C01827=1163.106,-119.094,-41.688,178.743,5.828,149.411
C01828=1163.100,-118.844,-41.697,178.746,5.829,149.411
C01829=1163.095,-118.594,-41.706,178.747,5.829,149.410
C01830=1163.090,-118.345,-41.714,178.749,5.829,149.410
C01831=1163.084,-118.095,-41.723,178.752,5.829,149.409
C01832=1163.079,-117.845,-41.731,178.754,5.830,149.409
C01833=1163.074,-117.595,-41.740,178.755,5.830,149.408
C01834=1163.068,-117.345,-41.749,178.758,5.830,149.408
C01835=1163.063,-117.095,-41.758,178.760,5.830,149.407
C01836=1163.058,-116.846,-41.766,178.762,5.831,149.407
C01837=1163.052,-116.596,-41.775,178.763,5.831,149.406
C01838=1163.047,-116.346,-41.784,178.766,5.831,149.405
C01839=1163.042,-116.097,-41.793,178.768,5.831,149.405
C01840=1163.036,-115.846,-41.803,178.770,5.832,149.404
C01841=1163.031,-115.597,-41.812,178.772,5.831,149.404
C01842=1163.025,-115.347,-41.820,178.774,5.832,149.403
C01843=1163.020,-115.098,-41.829,178.776,5.832,149.403
C01844=1163.015,-114.848,-41.838,178.778,5.833,149.402
C01845=1163.010,-114.598,-41.847,178.780,5.832,149.402
C01846=1163.005,-114.348,-41.856,178.782,5.833,149.401
C01847=1162.999,-114.098,-41.865,178.784,5.834,149.401
C01848=1162.993,-113.849,-41.874,178.786,5.834,149.400
C01849=1162.988,-113.599,-41.883,178.789,5.834,149.399
C01850=1162.983,-113.349,-41.891,178.790,5.834,149.399
C01851=1162.977,-113.099,-41.900,178.792,5.835,149.398
C01852=1162.972,-112.849,-41.909,178.795,5.835,149.398
C01853=1162.967,-112.600,-41.918,178.797,5.835,149.397
C01854=1162.961,-112.349,-41.928,178.798,5.835,149.397
C01855=1162.956,-112.099,-41.937,178.801,5.836,149.396
C01856=1162.950,-111.850,-41.945,178.803,5.836,149.395
C01857=1162.945,-111.600,-41.954,178.805,5.836,149.395
C01858=1162.940,-111.351,-41.963,178.808,5.837,149.394
C01859=1162.935,-111.101,-41.972,178.809,5.837,149.394
C01860=1162.929,-110.851,-41.982,178.811,5.838,149.393
C01861=1162.924,-110.601,-41.991,178.813,5.838,149.393
C01862=1162.919,-110.352,-42.000,178.816,5.838,149.392
C01863=1162.914,-110.102,-42.009,178.817,5.838,149.392
C01864=1162.908,-109.852,-42.018,178.819,5.839,149.391
C01865=1162.902,-109.602,-42.027,178.821,5.838,149.390
C01866=1162.897,-109.353,-42.036,178.824,5.839,149.390
C01867=1162.892,-109.103,-42.044,178.825,5.839,149.389
C01868=1162.887,-108.853,-42.054,178.828,5.839,149.389
C01869=1162.881,-108.603,-42.064,178.830,5.840,149.388
C01870=1162.876,-108.353,-42.072,178.832,5.840,149.388
C01871=1162.870,-108.104,-42.081,178.834,5.840,149.387
C01872=1162.865,-107.854,-42.090,178.836,5.840,149.387
C01873=1162.859,-107.604,-42.100,178.838,5.841,149.386
C01874=1162.855,-107.354,-42.109,178.840,5.841,149.385
C01875=1162.849,-107.104,-42.118,178.842,5.842,149.385
C01876=1162.844,-106.855,-42.127,178.845,5.842,149.384
C01877=1162.838,-106.604,-42.137,178.847,5.842,149.384
C01878=1162.833,-106.355,-42.146,178.849,5.843,149.383
C01879=1162.828,-106.105,-42.155,178.850,5.843,149.383
C01880=1162.823,-105.856,-42.164,178.853,5.843,149.382
C01881=1162.817,-105.606,-42.173,178.855,5.843,149.382
C01882=1162.811,-105.356,-42.182,178.857,5.844,149.381
C01883=1162.807,-105.107,-42.192,178.860,5.844,149.380
C01884=1162.801,-104.857,-42.201,178.861,5.844,149.380
C01885=1162.796,-104.607,-42.210,178.863,5.845,149.379
C01886=1162.790,-104.357,-42.219,178.866,5.844,149.379
C01887=1162.785,-104.108,-42.229,178.868,5.845,149.378
C01888=1162.780,-103.858,-42.238,178.869,5.845,149.378
C01889=1162.774,-103.608,-42.247,178.872,5.846,149.377
C01890=1162.769,-103.358,-42.256,178.874,5.846,149.376
C01891=1162.764,-103.108,-42.266,178.876,5.846,149.376
C01892=1162.758,-102.859,-42.275,178.878,5.847,149.375
C01893=1162.753,-102.587,-42.285,178.880,5.847,149.375
C01894=1162.747,-102.314,-42.296,178.883,5.847,149.374
C01895=1162.741,-102.043,-42.306,178.885,5.848,149.374
C01896=1162.735,-101.770,-42.316,178.888,5.848,149.373
C01897=1162.731,-101.521,-42.325,178.889,5.848,149.372
C01898=1162.725,-101.271,-42.335,178.892,5.848,149.372
C01899=1162.720,-101.021,-42.344,178.893,5.848,149.371
C01900=1162.715,-100.772,-42.353,178.896,5.849,149.371
C01901=1162.709,-100.521,-42.363,178.898,5.850,149.370
C01902=1162.704,-100.272,-42.373,178.900,5.850,149.369
C01903=1162.698,-100.022,-42.382,178.902,5.850,149.369
C01904=1162.693,-99.772,-42.391,178.904,5.850,149.368
C01905=1162.688,-99.523,-42.401,178.906,5.851,149.368
C01906=1162.682,-99.273,-42.410,178.908,5.851,149.367
C01907=1162.677,-99.024,-42.420,178.911,5.851,149.367
C01908=1162.671,-98.773,-42.429,178.913,5.852,149.366
C01909=1162.666,-98.523,-42.438,178.915,5.851,149.365
C01910=1162.661,-98.274,-42.448,178.917,5.852,149.365
C01911=1162.655,-98.024,-42.457,178.919,5.852,149.364
C01912=1162.651,-97.775,-42.467,178.921,5.853,149.364
C01913=1162.645,-97.525,-42.476,178.924,5.853,149.363
C01914=1162.640,-97.275,-42.486,178.925,5.853,149.363
C01915=1162.634,-97.025,-42.495,178.928,5.854,149.362
C01916=1162.629,-96.775,-42.504,178.929,5.854,149.362
C01917=1162.623,-96.526,-42.514,178.932,5.854,149.361
C01918=1162.619,-96.275,-42.524,178.934,5.855,149.360
C01919=1162.613,-96.026,-42.534,178.936,5.855,149.360
C01920=1162.608,-95.776,-42.543,178.939,5.855,149.359
C01921=1162.602,-95.526,-42.553,178.941,5.856,149.359
C01922=1162.597,-95.277,-42.562,178.942,5.856,149.358
C01923=1162.591,-95.027,-42.572,178.945,5.856,149.357
C01924=1162.586,-94.777,-42.581,178.947,5.856,149.357
C01925=1162.581,-94.528,-42.591,178.949,5.857,149.357
C01926=1162.575,-94.278,-42.600,178.952,5.857,149.356
C01927=1162.570,-94.028,-42.610,178.953,5.857,149.355
C01928=1162.565,-93.778,-42.620,178.956,5.858,149.355
C01929=1162.560,-93.528,-42.630,178.957,5.858,149.354
C01930=1162.555,-93.279,-42.639,178.960,5.859,149.354
C01931=1162.549,-93.029,-42.649,178.962,5.859,149.353
C01932=1162.544,-92.780,-42.659,178.964,5.859,149.352
C01933=1162.538,-92.529,-42.668,178.967,5.859,149.352
C01934=1162.533,-92.280,-42.678,178.969,5.860,149.351
C01935=1162.527,-92.030,-42.687,178.970,5.860,149.351
C01936=1162.523,-91.780,-42.697,178.973,5.860,149.350
C01937=1162.518,-91.530,-42.707,178.975,5.860,149.350
C01938=1162.512,-91.280,-42.717,178.977,5.861,149.349
C01939=1162.507,-91.031,-42.726,178.979,5.862,149.348
C01940=1162.501,-90.782,-42.737,178.981,5.862,149.348
C01941=1162.496,-90.532,-42.746,178.984,5.862,149.347
C01942=1162.491,-90.281,-42.756,178.986,5.863,149.347
C01943=1162.485,-90.031,-42.766,178.988,5.862,149.346
C01944=1162.480,-89.782,-42.775,178.990,5.863,149.346
C01945=1162.475,-89.533,-42.785,178.992,5.863,149.345
C01946=1162.469,-89.283,-42.794,178.994,5.863,149.344
C01947=1162.464,-89.033,-42.805,178.997,5.864,149.344
C01948=1162.459,-88.783,-42.815,178.999,5.864,149.343
C01949=1162.454,-88.533,-42.824,179.001,5.865,149.343
C01950=1162.448,-88.283,-42.834,179.003,5.865,149.342
C01951=1162.443,-88.034,-42.844,179.005,5.865,149.341
C01952=1162.438,-87.785,-42.854,179.007,5.866,149.341
C01953=1162.432,-87.534,-42.864,179.010,5.866,149.340
C01954=1162.427,-87.285,-42.874,179.012,5.866,149.340
C01955=1162.422,-87.035,-42.884,179.014,5.867,149.339
C01956=1162.416,-86.785,-42.893,179.017,5.867,149.339
C01957=1162.411,-86.536,-42.903,179.018,5.867,149.338
C01958=1162.406,-86.285,-42.913,179.021,5.868,149.337
C01959=1162.401,-86.036,-42.924,179.022,5.868,149.337
C01960=1162.395,-85.786,-42.933,179.025,5.868,149.336
C01961=1162.390,-85.536,-42.943,179.027,5.869,149.336
C01962=1162.385,-85.286,-42.953,179.029,5.869,149.335
C01963=1162.380,-85.037,-42.963,179.032,5.869,149.335
C01964=1162.374,-84.787,-42.973,179.034,5.870,149.334
C01965=1162.368,-84.537,-42.983,179.036,5.869,149.333
C01966=1162.364,-84.288,-42.992,179.038,5.870,149.333
C01967=1162.359,-84.038,-43.003,179.040,5.871,149.332
C01968=1162.353,-83.788,-43.013,179.042,5.871,149.332
C01969=1162.348,-83.539,-43.023,179.044,5.871,149.331
C01970=1162.343,-83.288,-43.032,179.047,5.872,149.330
C01971=1162.337,-83.039,-43.043,179.049,5.872,149.330
C01972=1162.332,-82.789,-43.053,179.051,5.873,149.330
C01973=1162.327,-82.540,-43.063,179.054,5.873,149.329
C01974=1162.322,-82.290,-43.073,179.055,5.873,149.328
C01975=1162.316,-82.040,-43.083,179.058,5.873,149.328
C01976=1162.311,-81.791,-43.094,179.060,5.874,149.327
C01977=1162.305,-81.541,-43.102,179.062,5.874,149.326
C01978=1162.300,-81.290,-43.113,179.064,5.874,149.326
C01979=1162.295,-81.041,-43.123,179.066,5.875,149.325
C01980=1162.289,-80.791,-43.133,179.069,5.875,149.325
C01981=1162.285,-80.541,-43.143,179.071,5.876,149.324
C01982=1162.279,-80.292,-43.154,179.073,5.876,149.324
C01983=1162.274,-80.042,-43.164,179.075,5.876,149.323
C01984=1162.268,-79.793,-43.174,179.078,5.876,149.322
C01985=1162.263,-79.543,-43.185,179.080,5.877,149.322
C01986=1162.258,-79.293,-43.194,179.081,5.877,149.321
C01987=1162.253,-79.044,-43.204,179.084,5.877,149.321
C01988=1162.248,-78.794,-43.215,179.086,5.878,149.320
C01989=1162.242,-78.544,-43.225,179.088,5.878,149.319
C01990=1162.236,-78.294,-43.235,179.091,5.879,149.319
C01991=1162.231,-78.044,-43.245,179.093,5.879,149.318
C01992=1162.226,-77.794,-43.255,179.095,5.880,149.318
C01993=1162.221,-77.545,-43.265,179.098,5.879,149.317
C01994=1162.216,-77.295,-43.276,179.100,5.880,149.317
C01995=1162.210,-77.045,-43.286,179.102,5.881,149.316
C01996=1162.205,-76.795,-43.296,179.104,5.881,149.315
C01997=1162.199,-76.524,-43.307,179.107,5.881,149.315
C01998=1162.194,-76.253,-43.319,179.109,5.882,149.314
C01999=1162.188,-75.983,-43.330,179.112,5.882,149.314
C02000=1162.182,-75.711,-43.341,179.114,5.883,149.313
C02001=1162.176,-75.461,-43.352,179.116,5.883,149.312
C02002=1162.171,-75.211,-43.362,179.118,5.883,149.312
C02003=1162.166,-74.962,-43.372,179.121,5.884,149.311
C02004=1162.160,-74.712,-43.383,179.122,5.884,149.311
C02005=1162.155,-74.462,-43.393,179.125,5.884,149.310
C02006=1162.150,-74.213,-43.403,179.127,5.885,149.309
C02007=1162.145,-73.962,-43.413,179.130,5.885,149.309
C02008=1162.140,-73.713,-43.424,179.131,5.885,149.308
C02009=1162.134,-73.463,-43.434,179.134,5.886,149.308
C02010=1162.129,-73.213,-43.444,179.136,5.886,149.307
C02011=1162.124,-72.964,-43.455,179.138,5.886,149.307
C02012=1162.118,-72.715,-43.465,179.140,5.887,149.306
C02013=1162.113,-72.464,-43.476,179.143,5.888,149.305
C02014=1162.108,-72.215,-43.486,179.145,5.888,149.305
C02015=1162.103,-71.965,-43.497,179.147,5.888,149.304
C02016=1162.097,-71.715,-43.507,179.150,5.888,149.304
C02017=1162.092,-71.465,-43.518,179.152,5.889,149.303
C02018=1162.087,-71.216,-43.529,179.154,5.889,149.302
C02019=1162.081,-70.966,-43.539,179.156,5.890,149.302
C02020=1162.076,-70.716,-43.549,179.159,5.890,149.301
C02021=1162.071,-70.467,-43.560,179.161,5.891,149.301
C02022=1162.066,-70.216,-43.570,179.163,5.890,149.300
C02023=1162.060,-69.967,-43.580,179.165,5.891,149.299
C02024=1162.055,-69.717,-43.592,179.167,5.892,149.299
C02025=1162.050,-69.468,-43.602,179.169,5.891,149.298
C02026=1162.044,-69.218,-43.612,179.172,5.892,149.298
C02027=1162.039,-68.968,-43.623,179.174,5.893,149.297
C02028=1162.034,-68.719,-43.634,179.177,5.893,149.297
C02029=1162.029,-68.469,-43.644,179.179,5.893,149.296
C02030=1162.023,-68.219,-43.654,179.181,5.894,149.295
C02031=1162.018,-67.969,-43.665,179.183,5.894,149.295
C02032=1162.013,-67.720,-43.676,179.186,5.895,149.294
C02033=1162.008,-67.470,-43.686,179.188,5.895,149.294
C02034=1162.002,-67.220,-43.697,179.190,5.895,149.293
C02035=1161.997,-66.970,-43.707,179.193,5.896,149.292
C02036=1161.992,-66.721,-43.718,179.194,5.896,149.292
C02037=1161.987,-66.471,-43.729,179.197,5.896,149.291
C02038=1161.981,-66.221,-43.739,179.199,5.897,149.291
C02039=1161.977,-65.972,-43.750,179.202,5.897,149.290
C02040=1161.971,-65.722,-43.760,179.203,5.897,149.290
C02041=1161.965,-65.471,-43.772,179.206,5.898,149.289
C02042=1161.960,-65.222,-43.782,179.208,5.899,149.288
C02043=1161.955,-64.972,-43.793,179.210,5.899,149.288
C02044=1161.950,-64.723,-43.803,179.212,5.899,149.287
C02045=1161.945,-64.473,-43.815,179.215,5.900,149.287
C02046=1161.939,-64.224,-43.825,179.217,5.900,149.286
C02047=1161.935,-63.974,-43.836,179.219,5.901,149.285
C02048=1161.929,-63.724,-43.846,179.222,5.900,149.285
C02049=1161.924,-63.474,-43.857,179.224,5.901,149.284
C02050=1161.918,-63.225,-43.868,179.226,5.902,149.284
C02051=1161.913,-62.975,-43.879,179.229,5.902,149.283
C02052=1161.908,-62.726,-43.890,179.231,5.902,149.282
C02053=1161.903,-62.475,-43.900,179.233,5.903,149.282
C02054=1161.897,-62.226,-43.911,179.236,5.903,149.281
C02055=1161.892,-61.976,-43.922,179.238,5.904,149.281
C02056=1161.887,-61.727,-43.932,179.240,5.904,149.280
C02057=1161.881,-61.477,-43.944,179.242,5.904,149.280
C02058=1161.876,-61.227,-43.955,179.245,5.905,149.279
C02059=1161.871,-60.978,-43.965,179.247,5.906,149.278
C02060=1161.866,-60.727,-43.976,179.249,5.906,149.278
C02061=1161.861,-60.478,-43.987,179.251,5.906,149.277
C02062=1161.855,-60.228,-43.998,179.254,5.906,149.276
C02063=1161.850,-59.978,-44.009,179.256,5.907,149.276
C02064=1161.845,-59.729,-44.020,179.259,5.908,149.275
C02065=1161.840,-59.479,-44.031,179.260,5.908,149.275
C02066=1161.834,-59.230,-44.041,179.263,5.908,149.274
C02067=1161.829,-58.980,-44.053,179.265,5.909,149.274
C02068=1161.823,-58.730,-44.063,179.268,5.909,149.273
C02069=1161.819,-58.480,-44.075,179.269,5.909,149.272
C02070=1161.814,-58.230,-44.085,179.272,5.910,149.272
C02071=1161.808,-57.981,-44.096,179.274,5.910,149.271
C02072=1161.803,-57.731,-44.107,179.277,5.911,149.271
C02073=1161.798,-57.481,-44.118,179.279,5.912,149.270
C02074=1161.792,-57.232,-44.129,179.281,5.911,149.269
C02075=1161.788,-56.982,-44.140,179.283,5.912,149.269
C02076=1161.782,-56.733,-44.152,179.286,5.912,149.268
C02077=1161.777,-56.482,-44.162,179.288,5.913,149.268
C02078=1161.772,-56.233,-44.173,179.291,5.914,149.267
C02079=1161.766,-55.983,-44.184,179.292,5.914,149.267
C02080=1161.761,-55.733,-44.195,179.295,5.914,149.266
C02081=1161.756,-55.484,-44.207,179.297,5.915,149.265
C02082=1161.751,-55.234,-44.217,179.300,5.915,149.265
C02083=1161.745,-54.984,-44.229,179.301,5.915,149.264
C02084=1161.741,-54.735,-44.240,179.304,5.916,149.263
C02085=1161.735,-54.485,-44.250,179.306,5.916,149.263
C02086=1161.730,-54.235,-44.262,179.309,5.917,149.262
C02087=1161.725,-53.986,-44.274,179.311,5.918,149.262
C02088=1161.719,-53.736,-44.284,179.313,5.917,149.261
C02089=1161.714,-53.486,-44.296,179.315,5.918,149.261
C02090=1161.709,-53.236,-44.307,179.318,5.918,149.260
C02091=1161.703,-52.987,-44.317,179.320,5.919,149.259
C02092=1161.698,-52.737,-44.329,179.323,5.920,149.259
C02093=1161.693,-52.487,-44.340,179.325,5.920,149.258
C02094=1161.688,-52.238,-44.351,179.327,5.920,149.258
C02095=1161.682,-51.988,-44.362,179.329,5.921,149.257
C02096=1161.678,-51.738,-44.374,179.332,5.921,149.256
C02097=1161.672,-51.489,-44.385,179.334,5.922,149.256
C02098=1161.667,-51.239,-44.396,179.337,5.922,149.255
C02099=1161.662,-50.989,-44.407,179.339,5.922,149.255
C02100=1161.657,-50.739,-44.419,179.341,5.923,149.254
C02101=1161.650,-50.469,-44.431,179.343,5.924,149.254
C02102=1161.646,-50.199,-44.443,179.346,5.924,149.253
C02103=1161.640,-49.928,-44.455,179.349,5.924,149.252
C02104=1161.634,-49.658,-44.467,179.351,5.925,149.251
C02105=1161.628,-49.408,-44.479,179.354,5.926,149.251
C02106=1161.624,-49.158,-44.491,179.356,5.926,149.250
C02107=1161.618,-48.909,-44.501,179.358,5.927,149.250
C02108=1161.613,-48.659,-44.513,179.361,5.926,149.249
C02109=1161.608,-48.409,-44.524,179.363,5.927,149.249
C02110=1161.603,-48.159,-44.536,179.365,5.928,149.248
C02111=1161.597,-47.910,-44.547,179.368,5.928,149.247
C02112=1161.592,-47.660,-44.559,179.370,5.929,149.247
C02113=1161.587,-47.411,-44.570,179.372,5.929,149.246
C02114=1161.581,-47.160,-44.581,179.374,5.929,149.246
C02115=1161.576,-46.911,-44.592,179.377,5.930,149.245
C02116=1161.571,-46.661,-44.604,179.379,5.931,149.244
C02117=1161.566,-46.411,-44.615,179.382,5.931,149.244
C02118=1161.561,-46.162,-44.627,179.384,5.932,149.243
C02119=1161.555,-45.913,-44.638,179.386,5.932,149.243
C02120=1161.550,-45.663,-44.650,179.388,5.932,149.242
C02121=1161.545,-45.413,-44.661,179.391,5.933,149.242
C02122=1161.540,-45.163,-44.673,179.393,5.933,149.241
C02123=1161.535,-44.913,-44.684,179.395,5.934,149.240
C02124=1161.529,-44.664,-44.696,179.398,5.935,149.240
C02125=1161.524,-44.415,-44.707,179.400,5.935,149.239
C02126=1161.519,-44.165,-44.719,179.402,5.935,149.238
C02127=1161.514,-43.915,-44.730,179.405,5.935,149.238
C02128=1161.509,-43.665,-44.742,179.407,5.936,149.237
C02129=1161.502,-43.415,-44.753,179.410,5.937,149.237
C02130=1161.498,-43.166,-44.764,179.412,5.937,149.236
C02131=1161.492,-42.916,-44.776,179.415,5.938,149.235
C02132=1161.488,-42.667,-44.788,179.417,5.939,149.235
C02133=1161.483,-42.417,-44.800,179.419,5.938,149.234
C02134=1161.478,-42.167,-44.811,179.421,5.939,149.234
C02135=1161.472,-41.918,-44.823,179.424,5.939,149.233
C02136=1161.466,-41.668,-44.835,179.426,5.940,149.233
C02137=1161.462,-41.418,-44.846,179.429,5.941,149.232
C02138=1161.456,-41.168,-44.858,179.431,5.941,149.231
C02139=1161.452,-40.919,-44.869,179.434,5.942,149.231
C02140=1161.446,-40.669,-44.881,179.435,5.942,149.230
C02141=1161.441,-40.419,-44.893,179.438,5.942,149.230
C02142=1161.435,-40.170,-44.904,179.440,5.943,149.229
C02143=1161.430,-39.920,-44.916,179.443,5.944,149.228
C02144=1161.425,-39.670,-44.928,179.445,5.944,149.228
C02145=1161.420,-39.420,-44.939,179.448,5.945,149.227
C02146=1161.414,-39.171,-44.951,179.450,5.945,149.226
C02147=1161.409,-38.921,-44.963,179.452,5.946,149.226
C02148=1161.405,-38.672,-44.975,179.454,5.946,149.225
C02149=1161.399,-38.422,-44.987,179.457,5.946,149.225
C02150=1161.393,-38.172,-44.998,179.459,5.947,149.224
C02151=1161.388,-37.923,-45.009,179.461,5.948,149.224
C02152=1161.383,-37.673,-45.021,179.464,5.948,149.223
C02153=1161.378,-37.423,-45.033,179.466,5.949,149.222
C02154=1161.373,-37.174,-45.045,179.469,5.949,149.222
C02155=1161.368,-36.924,-45.057,179.471,5.950,149.221
C02156=1161.362,-36.674,-45.069,179.473,5.950,149.221
C02157=1161.358,-36.424,-45.080,179.475,5.950,149.220
C02158=1161.352,-36.174,-45.092,179.478,5.951,149.219
C02159=1161.347,-35.925,-45.105,179.480,5.952,149.219
C02160=1161.342,-35.675,-45.117,179.483,5.952,149.218
C02161=1161.336,-35.426,-45.128,179.486,5.953,149.218
C02162=1161.331,-35.176,-45.139,179.488,5.953,149.217
C02163=1161.326,-34.927,-45.152,179.490,5.954,149.216
C02164=1161.320,-34.677,-45.164,179.493,5.955,149.216
C02165=1161.316,-34.428,-45.175,179.495,5.954,149.215
C02166=1161.310,-34.178,-45.187,179.497,5.955,149.215
C02167=1161.305,-33.928,-45.200,179.500,5.955,149.214
C02168=1161.300,-33.678,-45.212,179.502,5.956,149.214
C02169=1161.295,-33.429,-45.223,179.504,5.957,149.213
C02170=1161.290,-33.179,-45.235,179.507,5.957,149.212
C02171=1161.285,-32.929,-45.247,179.509,5.958,149.212
C02172=1161.279,-32.679,-45.259,179.511,5.959,149.211
C02173=1161.274,-32.430,-45.272,179.514,5.959,149.211
C02174=1161.269,-32.181,-45.283,179.516,5.960,149.210
C02175=1161.264,-31.931,-45.295,179.519,5.960,149.209
C02176=1161.259,-31.681,-45.308,179.521,5.960,149.209
C02177=1161.253,-31.431,-45.320,179.523,5.961,149.208
C02178=1161.248,-31.181,-45.331,179.526,5.961,149.208
C02179=1161.243,-30.932,-45.344,179.528,5.962,149.207
C02180=1161.238,-30.682,-45.355,179.531,5.962,149.206
C02181=1161.233,-30.433,-45.367,179.533,5.963,149.206
C02182=1161.227,-30.183,-45.380,179.535,5.964,149.205
C02183=1161.222,-29.933,-45.392,179.538,5.964,149.205
C02184=1161.217,-29.684,-45.404,179.540,5.965,149.204
C02185=1161.211,-29.434,-45.416,179.543,5.966,149.204
C02186=1161.207,-29.185,-45.428,179.545,5.966,149.203
C02187=1161.202,-28.935,-45.440,179.548,5.967,149.202
C02188=1161.196,-28.685,-45.452,179.550,5.967,149.202
C02189=1161.191,-28.436,-45.465,179.552,5.967,149.201
C02190=1161.186,-28.186,-45.476,179.554,5.968,149.200
C02191=1161.181,-27.937,-45.489,179.557,5.968,149.200
C02192=1161.175,-27.687,-45.501,179.559,5.969,149.199
C02193=1161.170,-27.437,-45.514,179.562,5.969,149.199
C02194=1161.165,-27.187,-45.525,179.564,5.970,149.198
C02195=1161.160,-26.937,-45.538,179.567,5.971,149.197
C02196=1161.155,-26.688,-45.550,179.569,5.971,149.197
C02197=1161.150,-26.438,-45.562,179.571,5.972,149.196
C02198=1161.145,-26.188,-45.574,179.574,5.973,149.196
C02199=1161.140,-25.939,-45.587,179.576,5.973,149.195
C02200=1161.134,-25.689,-45.599,179.579,5.974,149.194
C02201=1161.129,-25.440,-45.611,179.581,5.974,149.194
C02202=1161.124,-25.190,-45.623,179.584,5.975,149.193
C02203=1161.119,-24.941,-45.636,179.586,5.976,149.193
C02204=1161.113,-24.691,-45.648,179.589,5.976,149.192
C02205=1161.108,-24.421,-45.661,179.591,5.977,149.192
C02206=1161.102,-24.151,-45.676,179.593,5.977,149.191
C02207=1161.097,-23.881,-45.688,179.596,5.978,149.190
C02208=1161.091,-23.611,-45.701,179.599,5.978,149.190
C02209=1161.086,-23.362,-45.714,179.601,5.979,149.189
C02210=1161.081,-23.112,-45.726,179.604,5.979,149.188
C02211=1161.076,-22.862,-45.738,179.606,5.980,149.188
C02212=1161.070,-22.613,-45.751,179.609,5.981,149.187
C02213=1161.065,-22.364,-45.763,179.611,5.981,149.187
C02214=1161.060,-22.113,-45.776,179.613,5.982,149.186
C02215=1161.055,-21.864,-45.788,179.616,5.982,149.185
C02216=1161.050,-21.614,-45.801,179.618,5.983,149.185
C02217=1161.045,-21.365,-45.813,179.621,5.984,149.184
C02218=1161.039,-21.115,-45.826,179.623,5.984,149.184
C02219=1161.034,-20.866,-45.839,179.626,5.985,149.183
C02220=1161.028,-20.616,-45.850,179.628,5.986,149.183
C02221=1161.024,-20.366,-45.863,179.631,5.986,149.182
C02222=1161.019,-20.116,-45.876,179.633,5.987,149.181
C02223=1161.014,-19.867,-45.889,179.635,5.987,149.181
C02224=1161.008,-19.617,-45.900,179.638,5.988,149.180
C02225=1161.003,-19.368,-45.913,179.640,5.988,149.180
C02226=1160.999,-19.118,-45.926,179.642,5.988,149.179
C02227=1160.993,-18.868,-45.938,179.644,5.989,149.178
C02228=1160.988,-18.618,-45.951,179.647,5.989,149.178
C02229=1160.982,-18.369,-45.964,179.649,5.990,149.177
C02230=1160.977,-18.120,-45.976,179.652,5.991,149.176
C02231=1160.972,-17.870,-45.989,179.654,5.991,149.176
C02232=1160.967,-17.620,-46.001,179.657,5.992,149.175
C02233=1160.962,-17.370,-46.014,179.659,5.993,149.175
C02234=1160.957,-17.121,-46.026,179.662,5.993,149.174
C02235=1160.952,-16.872,-46.039,179.664,5.994,149.174
C02236=1160.946,-16.621,-46.053,179.666,5.994,149.173
C02237=1160.941,-16.372,-46.065,179.669,5.995,149.172
C02238=1160.936,-16.122,-46.077,179.671,5.996,149.172
C02239=1160.931,-15.873,-46.090,179.674,5.996,149.171
C02240=1160.926,-15.623,-46.102,179.676,5.997,149.171
C02241=1160.921,-15.373,-46.115,179.679,5.997,149.170
C02242=1160.915,-15.124,-46.128,179.681,5.998,149.170
C02243=1160.910,-14.874,-46.141,179.684,5.999,149.169
C02244=1160.905,-14.625,-46.154,179.686,5.999,149.168
C02245=1160.900,-14.375,-46.167,179.688,6.000,149.168
C02246=1160.895,-14.125,-46.178,179.691,6.000,149.167
C02247=1160.889,-13.876,-46.192,179.693,6.001,149.166
C02248=1160.884,-13.626,-46.204,179.696,6.002,149.166
C02249=1160.879,-13.376,-46.217,179.698,6.002,149.165
C02250=1160.874,-13.127,-46.230,179.701,6.003,149.165
C02251=1160.869,-12.877,-46.243,179.703,6.004,149.164
C02252=1160.864,-12.627,-46.256,179.706,6.004,149.163
C02253=1160.859,-12.378,-46.269,179.708,6.005,149.163
C02254=1160.854,-12.129,-46.281,179.711,6.006,149.162
C02255=1160.848,-11.879,-46.294,179.713,6.007,149.162
C02256=1160.843,-11.629,-46.307,179.716,6.007,149.161
C02257=1160.838,-11.380,-46.320,179.719,6.008,149.160
C02258=1160.833,-11.130,-46.333,179.721,6.009,149.160
C02259=1160.828,-10.880,-46.346,179.723,6.009,149.159
C02260=1160.823,-10.631,-46.359,179.726,6.010,149.159
C02261=1160.818,-10.381,-46.371,179.728,6.010,149.158
C02262=1160.812,-10.131,-46.385,179.730,6.011,149.158
C02263=1160.807,-9.882,-46.397,179.733,6.012,149.157
C02264=1160.802,-9.632,-46.410,179.735,6.012,149.157
C02265=1160.797,-9.382,-46.424,179.738,6.013,149.156
C02266=1160.792,-9.133,-46.436,179.741,6.013,149.155
C02267=1160.787,-8.884,-46.450,179.743,6.014,149.155
C02268=1160.782,-8.634,-46.463,179.745,6.015,149.154
C02269=1160.777,-8.384,-46.476,179.748,6.015,149.154
C02270=1160.771,-8.135,-46.488,179.750,6.016,149.153
C02271=1160.766,-7.885,-46.502,179.752,6.017,149.152
C02272=1160.761,-7.635,-46.514,179.755,6.017,149.152
C02273=1160.756,-7.385,-46.527,179.757,6.018,149.151
C02274=1160.751,-7.136,-46.541,179.760,6.018,149.151
C02275=1160.746,-6.887,-46.554,179.762,6.019,149.150
C02276=1160.741,-6.637,-46.567,179.765,6.020,149.149
C02277=1160.735,-6.387,-46.580,179.767,6.020,149.149
C02278=1160.730,-6.138,-46.593,179.770,6.021,149.148
C02279=1160.725,-5.888,-46.606,179.772,6.021,149.148
C02280=1160.720,-5.638,-46.619,179.775,6.023,149.147
C02281=1160.715,-5.389,-46.633,179.778,6.023,149.146
C02282=1160.710,-5.139,-46.646,179.780,6.024,149.146
C02283=1160.705,-4.890,-46.658,179.782,6.025,149.145
C02284=1160.699,-4.640,-46.672,179.785,6.025,149.145
C02285=1160.694,-4.390,-46.685,179.787,6.026,149.144
C02286=1160.689,-4.141,-46.699,179.789,6.027,149.144
C02287=1160.684,-3.891,-46.711,179.792,6.027,149.143
C02288=1160.678,-3.642,-46.725,179.795,6.028,149.142
C02289=1160.674,-3.392,-46.738,179.797,6.028,149.142
C02290=1160.668,-3.143,-46.751,179.800,6.029,149.141
C02291=1160.664,-2.893,-46.764,179.802,6.030,149.141
C02292=1160.658,-2.643,-46.778,179.804,6.030,149.140
C02293=1160.654,-2.394,-46.791,179.807,6.031,149.139
C02294=1160.649,-2.144,-46.804,179.810,6.032,149.139
C02295=1160.643,-1.894,-46.817,179.812,6.033,149.138
C02296=1160.638,-1.645,-46.831,179.815,6.033,149.138
C02297=1160.633,-1.396,-46.844,179.817,6.034,149.137
C02298=1160.627,-1.145,-46.858,179.820,6.035,149.136
C02299=1160.623,-0.897,-46.871,179.822,6.035,149.136
C02300=1160.617,-0.646,-46.884,179.824,6.036,149.135
C02301=1160.612,-0.397,-46.897,179.827,6.036,149.135
C02302=1160.607,-0.147,-46.911,179.829,6.037,149.134
C02303=1160.602,0.102,-46.924,179.832,6.038,149.133
C02304=1160.597,0.352,-46.937,179.834,6.039,149.133
C02305=1160.592,0.601,-46.951,179.837,6.039,149.132
C02306=1160.587,0.851,-46.964,179.839,6.041,149.132
C02307=1160.581,1.100,-46.978,179.842,6.041,149.131
C02308=1160.577,1.350,-46.991,179.844,6.042,149.131
C02309=1160.571,1.619,-47.006,179.847,6.042,149.130
C02310=1160.565,1.889,-47.020,179.850,6.043,149.129
C02311=1160.560,2.158,-47.035,179.853,6.044,149.129
C02312=1160.555,2.428,-47.050,179.855,6.045,149.128
C02313=1160.549,2.677,-47.063,179.858,6.045,149.127
C02314=1160.545,2.927,-47.076,179.860,6.046,149.127
C02315=1160.539,3.176,-47.090,179.862,6.047,149.126
C02316=1160.534,3.426,-47.104,179.865,6.047,149.126
C02317=1160.529,3.675,-47.116,179.867,6.048,149.125
C02318=1160.524,3.925,-47.131,179.870,6.048,149.124
C02319=1160.518,4.175,-47.144,179.873,6.050,149.124
C02320=1160.514,4.424,-47.158,179.875,6.050,149.123
C02321=1160.508,4.674,-47.171,179.878,6.051,149.123
C02322=1160.503,4.923,-47.185,179.880,6.052,149.122
C02323=1160.499,5.173,-47.199,179.882,6.053,149.122
C02324=1160.493,5.422,-47.212,179.885,6.053,149.121
C02325=1160.488,5.672,-47.226,179.888,6.053,149.120
C02326=1160.483,5.921,-47.239,179.890,6.054,149.120
C02327=1160.478,6.171,-47.253,179.893,6.055,149.119
C02328=1160.473,6.421,-47.267,179.895,6.056,149.119
C02329=1160.468,6.670,-47.280,179.898,6.057,149.118
C02330=1160.463,6.920,-47.294,179.900,6.058,149.118
C02331=1160.457,7.169,-47.307,179.903,6.058,149.117
C02332=1160.453,7.419,-47.321,179.905,6.059,149.116
C02333=1160.448,7.669,-47.335,179.908,6.059,149.116
C02334=1160.442,7.918,-47.349,179.910,6.060,149.115
C02335=1160.437,8.168,-47.363,179.913,6.061,149.115
C02336=1160.432,8.417,-47.376,179.915,6.062,149.114
C02337=1160.427,8.667,-47.390,179.918,6.063,149.113
C02338=1160.422,8.917,-47.404,179.920,6.063,149.113
C02339=1160.416,9.166,-47.418,179.923,6.064,149.112
C02340=1160.412,9.416,-47.431,179.925,6.064,149.112
C02341=1160.407,9.665,-47.445,179.927,6.065,149.111
C02342=1160.401,9.914,-47.459,179.931,6.067,149.110
C02343=1160.396,10.165,-47.473,179.933,6.067,149.110
C02344=1160.390,10.414,-47.487,179.935,6.068,149.109
C02345=1160.386,10.663,-47.500,179.938,6.069,149.109
C02346=1160.381,10.913,-47.515,179.940,6.069,149.108
C02347=1160.375,11.162,-47.528,179.942,6.070,149.108
C02348=1160.370,11.412,-47.542,179.946,6.071,149.107
C02349=1160.366,11.662,-47.556,179.948,6.072,149.107
C02350=1160.360,11.911,-47.570,179.951,6.072,149.106
C02351=1160.356,12.160,-47.584,179.953,6.073,149.105
C02352=1160.350,12.411,-47.597,179.955,6.074,149.105
C02353=1160.345,12.660,-47.611,179.958,6.074,149.104
C02354=1160.340,12.909,-47.626,179.961,6.076,149.104
C02355=1160.335,13.159,-47.640,179.963,6.076,149.103
C02356=1160.330,13.409,-47.654,179.966,6.077,149.102
C02357=1160.325,13.658,-47.668,179.968,6.078,149.102
C02358=1160.320,13.908,-47.681,179.970,6.078,149.101
C02359=1160.315,14.158,-47.695,179.973,6.079,149.101
C02360=1160.309,14.407,-47.709,179.976,6.081,149.100
C02361=1160.305,14.656,-47.724,179.978,6.081,149.100
C02362=1160.300,14.906,-47.738,179.981,6.082,149.099
C02363=1160.295,15.156,-47.752,179.983,6.082,149.098
C02364=1160.289,15.405,-47.766,179.986,6.083,149.098
C02365=1160.284,15.654,-47.780,179.988,6.084,149.097
C02366=1160.279,15.904,-47.795,179.991,6.085,149.097
C02367=1160.274,16.153,-47.808,179.994,6.086,149.096
C02368=1160.268,16.403,-47.822,179.996,6.086,149.095
C02369=1160.263,16.653,-47.836,179.998,6.087,149.095
C02370=1160.258,16.903,-47.851,-179.999,6.087,149.094
C02371=1160.254,17.152,-47.864,-179.996,6.089,149.094
C02372=1160.249,17.401,-47.878,-179.994,6.090,149.093
C02373=1160.244,17.651,-47.892,-179.991,6.090,149.093
C02374=1160.239,17.901,-47.907,-179.989,6.091,149.092
C02375=1160.234,18.150,-47.921,-179.987,6.092,149.092
C02376=1160.228,18.399,-47.935,-179.983,6.093,149.091
C02377=1160.223,18.649,-47.949,-179.981,6.094,149.090
C02378=1160.218,18.899,-47.963,-179.979,6.094,149.090
C02379=1160.213,19.149,-47.978,-179.976,6.095,149.089
C02380=1160.208,19.398,-47.992,-179.974,6.096,149.089
C02381=1160.203,19.647,-48.007,-179.970,6.097,149.088
C02382=1160.198,19.896,-48.021,-179.968,6.098,149.087
C02383=1160.193,20.146,-48.036,-179.966,6.098,149.087
C02384=1160.188,20.396,-48.050,-179.964,6.099,149.086
C02385=1160.183,20.646,-48.064,-179.961,6.099,149.086
C02386=1160.177,20.895,-48.078,-179.958,6.101,149.085
C02387=1160.172,21.145,-48.093,-179.955,6.102,149.084
C02388=1160.167,21.394,-48.107,-179.953,6.102,149.084
C02389=1160.162,21.644,-48.121,-179.951,6.103,149.083
C02390=1160.157,21.894,-48.135,-179.948,6.104,149.083
C02391=1160.153,22.143,-48.150,-179.945,6.105,149.082
C02392=1160.147,22.392,-48.164,-179.943,6.106,149.082
C02393=1160.142,22.641,-48.179,-179.940,6.106,149.081
C02394=1160.137,22.891,-48.193,-179.938,6.107,149.081
C02395=1160.132,23.141,-48.207,-179.935,6.108,149.080
C02396=1160.126,23.391,-48.222,-179.933,6.109,149.079
C02397=1160.122,23.640,-48.237,-179.930,6.110,149.079
C02398=1160.117,23.890,-48.251,-179.928,6.110,149.078
C02399=1160.111,24.139,-48.265,-179.925,6.112,149.078
C02400=1160.106,24.388,-48.279,-179.923,6.113,149.077
C02401=1160.102,24.638,-48.294,-179.920,6.113,149.077
C02402=1160.097,24.887,-48.309,-179.918,6.114,149.076
C02403=1160.091,25.137,-48.324,-179.915,6.115,149.075
C02404=1160.086,25.387,-48.338,-179.912,6.116,149.075
C02405=1160.081,25.636,-48.353,-179.910,6.116,149.074
C02406=1160.076,25.886,-48.367,-179.907,6.117,149.074
C02407=1160.072,26.135,-48.381,-179.904,6.119,149.073
C02408=1160.066,26.384,-48.395,-179.902,6.119,149.072
C02409=1160.061,26.634,-48.411,-179.900,6.120,149.072
C02410=1160.056,26.884,-48.425,-179.897,6.120,149.071
C02411=1160.051,27.133,-48.439,-179.894,6.122,149.071
C02412=1160.046,27.382,-48.454,-179.891,6.122,149.070
C02413=1160.040,27.651,-48.471,-179.889,6.123,149.070
C02414=1160.035,27.921,-48.486,-179.886,6.125,149.069
C02415=1160.030,28.190,-48.501,-179.883,6.125,149.068
C02416=1160.024,28.459,-48.518,-179.881,6.127,149.068
C02417=1160.019,28.708,-48.533,-179.878,6.127,149.067
C02418=1160.014,28.958,-48.547,-179.876,6.128,149.067
C02419=1160.009,29.207,-48.561,-179.873,6.129,149.066
C02420=1160.004,29.457,-48.577,-179.870,6.130,149.065
C02421=1159.999,29.706,-48.591,-179.868,6.131,149.065
C02422=1159.994,29.956,-48.606,-179.865,6.131,149.064
C02423=1159.989,30.205,-48.620,-179.863,6.132,149.064
C02424=1159.984,30.455,-48.636,-179.860,6.133,149.063
C02425=1159.979,30.704,-48.650,-179.858,6.134,149.063
C02426=1159.974,30.954,-48.665,-179.855,6.135,149.062
C02427=1159.968,31.203,-48.680,-179.852,6.136,149.062
C02428=1159.963,31.452,-48.694,-179.850,6.137,149.061
C02429=1159.958,31.702,-48.709,-179.847,6.138,149.060
C02430=1159.953,31.952,-48.724,-179.845,6.138,149.060
C02431=1159.949,32.201,-48.739,-179.842,6.140,149.059
C02432=1159.944,32.451,-48.754,-179.839,6.140,149.059
C02433=1159.938,32.700,-48.769,-179.837,6.141,149.058
C02434=1159.934,32.950,-48.784,-179.834,6.142,149.058
C02435=1159.929,33.199,-48.798,-179.832,6.143,149.057
C02436=1159.923,33.449,-48.814,-179.829,6.144,149.056
C02437=1159.918,33.698,-48.828,-179.827,6.144,149.056
C02438=1159.913,33.948,-48.844,-179.824,6.146,149.055
C02439=1159.908,34.198,-48.858,-179.822,6.147,149.055
C02440=1159.903,34.447,-48.873,-179.819,6.147,149.054
C02441=1159.898,34.697,-48.888,-179.816,6.149,149.054
C02442=1159.893,34.946,-48.903,-179.814,6.149,149.053
C02443=1159.888,35.195,-48.919,-179.811,6.150,149.053
C02444=1159.883,35.445,-48.933,-179.808,6.151,149.052
C02445=1159.878,35.694,-48.948,-179.806,6.152,149.051
C02446=1159.873,35.943,-48.963,-179.803,6.153,149.051
C02447=1159.868,36.193,-48.978,-179.801,6.154,149.050
C02448=1159.862,36.442,-48.993,-179.798,6.155,149.050
C02449=1159.858,36.692,-49.008,-179.796,6.156,149.049
C02450=1159.852,36.942,-49.023,-179.793,6.156,149.049
C02451=1159.848,37.191,-49.039,-179.790,6.158,149.048
C02452=1159.843,37.441,-49.054,-179.788,6.158,149.047
C02453=1159.838,37.690,-49.068,-179.786,6.159,149.047
C02454=1159.832,37.940,-49.084,-179.782,6.160,149.046
C02455=1159.828,38.189,-49.099,-179.780,6.161,149.046
C02456=1159.822,38.438,-49.115,-179.778,6.162,149.045
C02457=1159.817,38.688,-49.129,-179.775,6.163,149.045
C02458=1159.812,38.937,-49.144,-179.773,6.164,149.044
C02459=1159.807,39.187,-49.159,-179.770,6.165,149.044
C02460=1159.802,39.436,-49.175,-179.767,6.166,149.043
C02461=1159.797,39.686,-49.190,-179.765,6.167,149.043
C02462=1159.792,39.936,-49.205,-179.762,6.168,149.042
C02463=1159.787,40.185,-49.220,-179.759,6.169,149.041
C02464=1159.782,40.434,-49.236,-179.757,6.170,149.041
C02465=1159.777,40.683,-49.251,-179.754,6.170,149.040
C02466=1159.772,40.933,-49.266,-179.752,6.172,149.040
C02467=1159.767,41.183,-49.282,-179.749,6.172,149.039
C02468=1159.762,41.433,-49.297,-179.747,6.173,149.039
C02469=1159.757,41.682,-49.312,-179.744,6.174,149.038
C02470=1159.752,41.931,-49.327,-179.741,6.175,149.038
C02471=1159.747,42.180,-49.343,-179.739,6.176,149.037
C02472=1159.742,42.430,-49.357,-179.736,6.177,149.036
C02473=1159.737,42.680,-49.373,-179.733,6.178,149.036
C02474=1159.732,42.930,-49.389,-179.731,6.180,149.035
C02475=1159.727,43.179,-49.404,-179.728,6.180,149.035
C02476=1159.722,43.428,-49.419,-179.726,6.181,149.034
C02477=1159.716,43.678,-49.435,-179.723,6.182,149.034
C02478=1159.712,43.927,-49.450,-179.720,6.183,149.033
C02479=1159.707,44.177,-49.466,-179.718,6.184,149.032
C02480=1159.701,44.426,-49.481,-179.715,6.185,149.032
C02481=1159.697,44.675,-49.496,-179.712,6.186,149.031
C02482=1159.691,44.925,-49.512,-179.710,6.187,149.031
C02483=1159.687,45.174,-49.527,-179.707,6.188,149.030
C02484=1159.682,45.424,-49.543,-179.705,6.189,149.030
C02485=1159.677,45.673,-49.558,-179.702,6.190,149.029
C02486=1159.671,45.923,-49.574,-179.700,6.191,149.029
C02487=1159.667,46.172,-49.589,-179.697,6.192,149.028
C02488=1159.662,46.422,-49.605,-179.694,6.193,149.028
C02489=1159.656,46.671,-49.621,-179.692,6.194,149.027
C02490=1159.652,46.920,-49.636,-179.689,6.194,149.026
C02491=1159.647,47.170,-49.652,-179.687,6.196,149.026
C02492=1159.642,47.420,-49.667,-179.684,6.196,149.025
C02493=1159.636,47.669,-49.683,-179.681,6.198,149.025
C02494=1159.631,47.918,-49.698,-179.679,6.199,149.024
C02495=1159.627,48.168,-49.714,-179.676,6.199,149.024
C02496=1159.621,48.418,-49.729,-179.673,6.201,149.023
C02497=1159.616,48.667,-49.746,-179.671,6.202,149.023
C02498=1159.612,48.916,-49.761,-179.668,6.203,149.022
C02499=1159.607,49.166,-49.777,-179.666,6.204,149.022
C02500=1159.601,49.415,-49.792,-179.663,6.205,149.021
C02501=1159.597,49.665,-49.808,-179.660,6.206,149.020
C02502=1159.592,49.914,-49.823,-179.658,6.207,149.020
C02503=1159.587,50.164,-49.839,-179.655,6.208,149.019
C02504=1159.582,50.413,-49.855,-179.653,6.209,149.019
C02505=1159.577,50.663,-49.871,-179.650,6.209,149.018
C02506=1159.571,50.912,-49.886,-179.647,6.211,149.018
C02507=1159.567,51.162,-49.902,-179.645,6.212,149.017
C02508=1159.562,51.411,-49.917,-179.642,6.213,149.017
C02509=1159.557,51.660,-49.934,-179.639,6.214,149.016
C02510=1159.552,51.910,-49.950,-179.637,6.215,149.016
C02511=1159.547,52.160,-49.965,-179.634,6.216,149.015
C02512=1159.541,52.409,-49.981,-179.632,6.217,149.014
C02513=1159.537,52.658,-49.998,-179.629,6.218,149.014
C02514=1159.532,52.908,-50.013,-179.626,6.219,149.013
C02515=1159.527,53.157,-50.028,-179.624,6.220,149.013
C02516=1159.522,53.406,-50.045,-179.621,6.221,149.012
C02517=1159.517,53.675,-50.062,-179.618,6.223,149.012
C02518=1159.511,53.943,-50.079,-179.616,6.223,149.011
C02519=1159.506,54.212,-50.096,-179.612,6.224,149.010
C02520=1159.501,54.481,-50.113,-179.610,6.225,149.010
C02521=1159.495,54.730,-50.129,-179.607,6.227,149.009
C02522=1159.490,54.980,-50.144,-179.605,6.227,149.009
C02523=1159.485,55.229,-50.161,-179.602,6.229,149.008
C02524=1159.480,55.479,-50.177,-179.599,6.230,149.008
C02525=1159.476,55.728,-50.193,-179.596,6.231,149.007
C02526=1159.470,55.978,-50.209,-179.594,6.232,149.007
C02527=1159.465,56.227,-50.224,-179.592,6.233,149.006
C02528=1159.460,56.477,-50.241,-179.589,6.234,149.006
C02529=1159.455,56.726,-50.257,-179.587,6.235,149.005
C02530=1159.450,56.975,-50.273,-179.583,6.236,149.004
C02531=1159.445,57.225,-50.289,-179.581,6.237,149.004
C02532=1159.440,57.475,-50.305,-179.578,6.238,149.003
C02533=1159.435,57.724,-50.321,-179.576,6.239,149.003
C02534=1159.430,57.973,-50.337,-179.573,6.240,149.002
C02535=1159.425,58.223,-50.354,-179.570,6.241,149.002
C02536=1159.420,58.472,-50.369,-179.568,6.242,149.001
C02537=1159.415,58.722,-50.386,-179.565,6.243,149.001
C02538=1159.410,58.971,-50.401,-179.563,6.244,149.000
C02539=1159.406,59.220,-50.418,-179.560,6.246,149.000
C02540=1159.400,59.470,-50.434,-179.557,6.246,148.999
C02541=1159.396,59.719,-50.450,-179.554,6.248,148.999
C02542=1159.390,59.969,-50.466,-179.552,6.249,148.998
C02543=1159.386,60.218,-50.483,-179.549,6.250,148.998
C02544=1159.381,60.467,-50.499,-179.547,6.251,148.997
C02545=1159.376,60.717,-50.515,-179.544,6.252,148.997
C02546=1159.371,60.966,-50.531,-179.541,6.253,148.996
C02547=1159.366,61.216,-50.547,-179.539,6.255,148.995
C02548=1159.361,61.465,-50.563,-179.536,6.255,148.995
C02549=1159.356,61.715,-50.581,-179.533,6.257,148.994
C02550=1159.350,61.964,-50.596,-179.531,6.258,148.994
C02551=1159.346,62.213,-50.613,-179.528,6.259,148.993
C02552=1159.341,62.463,-50.628,-179.526,6.260,148.993
C02553=1159.336,62.712,-50.645,-179.523,6.260,148.992
C02554=1159.331,62.961,-50.661,-179.520,6.262,148.992
C02555=1159.326,63.211,-50.677,-179.518,6.263,148.991
C02556=1159.321,63.460,-50.694,-179.515,6.264,148.991
C02557=1159.316,63.710,-50.711,-179.513,6.265,148.990
C02558=1159.311,63.960,-50.727,-179.510,6.266,148.990
C02559=1159.306,64.209,-50.743,-179.507,6.267,148.989
C02560=1159.302,64.458,-50.760,-179.504,6.269,148.988
C02561=1159.296,64.707,-50.776,-179.502,6.269,148.988
C02562=1159.292,64.957,-50.792,-179.499,6.271,148.988
C02563=1159.286,65.206,-50.809,-179.497,6.272,148.987
C02564=1159.281,65.456,-50.826,-179.494,6.273,148.986
C02565=1159.277,65.705,-50.842,-179.491,6.274,148.986
C02566=1159.271,65.954,-50.858,-179.489,6.275,148.985
C02567=1159.266,66.204,-50.875,-179.486,6.276,148.985
C02568=1159.261,66.453,-50.892,-179.483,6.278,148.984
C02569=1159.257,66.703,-50.908,-179.481,6.278,148.984
C02570=1159.252,66.952,-50.925,-179.478,6.280,148.983
C02571=1159.247,67.201,-50.940,-179.475,6.281,148.983
C02572=1159.242,67.451,-50.958,-179.473,6.282,148.982
C02573=1159.237,67.700,-50.974,-179.470,6.284,148.982
C02574=1159.232,67.949,-50.991,-179.468,6.284,148.981
C02575=1159.227,68.199,-51.008,-179.464,6.286,148.981
C02576=1159.222,68.448,-51.024,-179.462,6.287,148.980
C02577=1159.217,68.698,-51.041,-179.459,6.288,148.980
C02578=1159.212,68.948,-51.057,-179.457,6.289,148.979
C02579=1159.207,69.197,-51.074,-179.454,6.291,148.979
C02580=1159.202,69.446,-51.090,-179.451,6.291,148.978
C02581=1159.198,69.696,-51.107,-179.449,6.293,148.978
C02582=1159.192,69.945,-51.124,-179.447,6.294,148.977
C02583=1159.187,70.194,-51.141,-179.443,6.295,148.976
C02584=1159.183,70.444,-51.157,-179.441,6.296,148.976
C02585=1159.177,70.693,-51.174,-179.438,6.297,148.975
C02586=1159.173,70.942,-51.191,-179.436,6.298,148.975
C02587=1159.168,71.192,-51.208,-179.433,6.300,148.974
C02588=1159.162,71.441,-51.225,-179.430,6.301,148.974
C02589=1159.158,71.690,-51.241,-179.428,6.302,148.973
C02590=1159.153,71.940,-51.258,-179.424,6.303,148.973
C02591=1159.148,72.189,-51.275,-179.422,6.304,148.972
C02592=1159.143,72.438,-51.291,-179.420,6.306,148.972
C02593=1159.138,72.688,-51.309,-179.417,6.306,148.971
C02594=1159.133,72.938,-51.325,-179.414,6.308,148.971
C02595=1159.128,73.187,-51.342,-179.412,6.308,148.970
C02596=1159.123,73.436,-51.359,-179.409,6.310,148.970
C02597=1159.119,73.686,-51.376,-179.406,6.312,148.969
C02598=1159.113,73.935,-51.392,-179.404,6.312,148.969
C02599=1159.108,74.184,-51.409,-179.401,6.314,148.968
C02600=1159.103,74.434,-51.426,-179.399,6.315,148.968
C02601=1159.099,74.683,-51.444,-179.395,6.316,148.967
C02602=1159.093,74.932,-51.461,-179.393,6.317,148.967
C02603=1159.089,75.182,-51.477,-179.390,6.318,148.966
C02604=1159.083,75.431,-51.495,-179.388,6.319,148.966
C02605=1159.079,75.681,-51.511,-179.385,6.321,148.965
C02606=1159.074,75.931,-51.529,-179.382,6.322,148.965
C02607=1159.069,76.179,-51.546,-179.380,6.323,148.964
C02608=1159.064,76.429,-51.563,-179.377,6.325,148.964
C02609=1159.059,76.678,-51.580,-179.374,6.325,148.963
C02610=1159.054,76.928,-51.597,-179.372,6.327,148.963
C02611=1159.049,77.177,-51.613,-179.369,6.329,148.962
C02612=1159.044,77.426,-51.631,-179.366,6.329,148.961
C02613=1159.040,77.675,-51.648,-179.364,6.331,148.961
C02614=1159.034,77.925,-51.665,-179.361,6.331,148.960
C02615=1159.030,78.175,-51.682,-179.358,6.333,148.960
C02616=1159.024,78.423,-51.699,-179.356,6.334,148.960
C02617=1159.019,78.673,-51.717,-179.353,6.335,148.959
C02618=1159.015,78.922,-51.733,-179.350,6.337,148.958
C02619=1159.009,79.172,-51.750,-179.348,6.338,148.958
C02620=1159.005,79.421,-51.768,-179.345,6.339,148.957
C02621=1158.999,79.689,-51.786,-179.342,6.341,148.957
C02622=1158.994,79.958,-51.805,-179.339,6.341,148.956
C02623=1158.989,80.227,-51.823,-179.337,6.343,148.956
C02624=1158.984,80.494,-51.842,-179.333,6.344,148.955
C02625=1158.978,80.744,-51.859,-179.331,6.346,148.955
C02626=1158.974,80.994,-51.876,-179.328,6.346,148.954
C02627=1158.969,81.243,-51.894,-179.325,6.348,148.954
C02628=1158.964,81.492,-51.911,-179.323,6.350,148.953
C02629=1158.959,81.742,-51.928,-179.320,6.350,148.953
C02630=1158.954,81.991,-51.946,-179.317,6.352,148.952
C02631=1158.948,82.240,-51.963,-179.315,6.353,148.952
C02632=1158.944,82.489,-51.980,-179.312,6.354,148.951
C02633=1158.939,82.739,-51.997,-179.309,6.356,148.951
C02634=1158.934,82.988,-52.015,-179.307,6.357,148.950
C02635=1158.930,83.238,-52.032,-179.304,6.358,148.950
C02636=1158.924,83.487,-52.049,-179.302,6.359,148.949
C02637=1158.920,83.737,-52.067,-179.299,6.361,148.949
C02638=1158.915,83.986,-52.084,-179.296,6.362,148.948
C02639=1158.910,84.235,-52.102,-179.294,6.363,148.948
C02640=1158.905,84.485,-52.119,-179.291,6.365,148.947
C02641=1158.900,84.734,-52.137,-179.288,6.366,148.947
C02642=1158.895,84.983,-52.153,-179.285,6.367,148.946
C02643=1158.890,85.232,-52.171,-179.283,6.368,148.946
C02644=1158.885,85.481,-52.189,-179.280,6.370,148.945
C02645=1158.880,85.731,-52.207,-179.277,6.371,148.945
C02646=1158.876,85.980,-52.224,-179.275,6.372,148.944
C02647=1158.871,86.230,-52.241,-179.272,6.373,148.944
C02648=1158.866,86.479,-52.259,-179.269,6.374,148.943
C02649=1158.860,86.729,-52.277,-179.267,6.376,148.943
C02650=1158.856,86.978,-52.294,-179.264,6.377,148.942
C02651=1158.851,87.227,-52.312,-179.261,6.378,148.942
C02652=1158.846,87.477,-52.329,-179.258,6.380,148.941
C02653=1158.841,87.726,-52.347,-179.256,6.381,148.941
C02654=1158.836,87.975,-52.365,-179.253,6.382,148.940
C02655=1158.831,88.225,-52.382,-179.250,6.384,148.940
C02656=1158.827,88.474,-52.400,-179.248,6.384,148.939
C02657=1158.822,88.723,-52.418,-179.245,6.386,148.939
C02658=1158.817,88.973,-52.435,-179.242,6.388,148.938
C02659=1158.812,89.222,-52.453,-179.240,6.388,148.938
C02660=1158.807,89.471,-52.471,-179.237,6.390,148.937
C02661=1158.802,89.721,-52.488,-179.234,6.392,148.937
C02662=1158.797,89.970,-52.506,-179.232,6.393,148.936
C02663=1158.793,90.219,-52.524,-179.229,6.394,148.936
C02664=1158.788,90.468,-52.542,-179.226,6.396,148.935
C02665=1158.782,90.718,-52.559,-179.224,6.397,148.935
C02666=1158.778,90.967,-52.577,-179.221,6.398,148.934
C02667=1158.773,91.216,-52.595,-179.218,6.400,148.934
C02668=1158.768,91.465,-52.613,-179.216,6.400,148.933
C02669=1158.763,91.714,-52.631,-179.213,6.402,148.933
C02670=1158.758,91.964,-52.648,-179.210,6.403,148.932
C02671=1158.753,92.213,-52.666,-179.207,6.405,148.932
C02672=1158.748,92.463,-52.684,-179.205,6.406,148.932
C02673=1158.743,92.712,-52.702,-179.202,6.407,148.931
C02674=1158.739,92.962,-52.720,-179.199,6.409,148.930
C02675=1158.734,93.211,-52.738,-179.197,6.410,148.930
C02676=1158.728,93.461,-52.756,-179.194,6.411,148.929
C02677=1158.724,93.710,-52.774,-179.191,6.413,148.929
C02678=1158.719,93.959,-52.792,-179.189,6.414,148.929
C02679=1158.714,94.208,-52.810,-179.186,6.415,148.928
C02680=1158.709,94.457,-52.828,-179.183,6.417,148.928
C02681=1158.704,94.706,-52.846,-179.181,6.418,148.927
C02682=1158.700,94.956,-52.864,-179.178,6.419,148.927
C02683=1158.695,95.206,-52.882,-179.175,6.421,148.926
C02684=1158.690,95.455,-52.900,-179.172,6.423,148.926
C02685=1158.685,95.704,-52.918,-179.170,6.423,148.925
C02686=1158.680,95.953,-52.936,-179.167,6.425,148.925
C02687=1158.675,96.202,-52.954,-179.164,6.426,148.924
C02688=1158.670,96.451,-52.972,-179.162,6.427,148.924
C02689=1158.665,96.701,-52.990,-179.159,6.429,148.923
C02690=1158.661,96.950,-53.008,-179.156,6.430,148.923
C02691=1158.656,97.200,-53.026,-179.153,6.432,148.922
C02692=1158.651,97.449,-53.044,-179.151,6.433,148.922
C02693=1158.646,97.698,-53.062,-179.148,6.435,148.921
C02694=1158.640,97.947,-53.081,-179.145,6.436,148.921
C02695=1158.636,98.197,-53.099,-179.143,6.438,148.920
C02696=1158.631,98.447,-53.117,-179.140,6.439,148.920
C02697=1158.626,98.696,-53.135,-179.137,6.440,148.919
C02698=1158.621,98.945,-53.153,-179.134,6.442,148.919
C02699=1158.617,99.194,-53.171,-179.132,6.442,148.918
C02700=1158.612,99.443,-53.189,-179.130,6.444,148.918
C02701=1158.608,99.692,-53.208,-179.126,6.445,148.917
C02702=1158.602,99.942,-53.226,-179.124,6.447,148.917
C02703=1158.597,100.191,-53.244,-179.122,6.448,148.917
C02704=1158.592,100.440,-53.262,-179.119,6.450,148.916
C02705=1158.587,100.689,-53.280,-179.116,6.451,148.916
C02706=1158.583,100.939,-53.299,-179.113,6.453,148.915
C02707=1158.578,101.188,-53.318,-179.111,6.454,148.915
C02708=1158.573,101.437,-53.336,-179.108,6.455,148.914
C02709=1158.568,101.687,-53.354,-179.105,6.457,148.914
C02710=1158.563,101.936,-53.372,-179.102,6.458,148.913
C02711=1158.559,102.186,-53.390,-179.100,6.459,148.913
C02712=1158.553,102.434,-53.410,-179.097,6.461,148.912
C02713=1158.548,102.684,-53.428,-179.094,6.462,148.912
C02714=1158.544,102.934,-53.446,-179.091,6.464,148.911
C02715=1158.539,103.183,-53.464,-179.089,6.466,148.911
C02716=1158.534,103.432,-53.483,-179.086,6.467,148.911
C02717=1158.529,103.681,-53.501,-179.083,6.468,148.910
C02718=1158.524,103.931,-53.520,-179.081,6.470,148.909
C02719=1158.519,104.179,-53.539,-179.078,6.471,148.909
C02720=1158.514,104.429,-53.557,-179.076,6.472,148.909
C02721=1158.510,104.679,-53.575,-179.072,6.474,148.908
C02722=1158.505,104.927,-53.594,-179.070,6.475,148.908
C02723=1158.500,105.177,-53.612,-179.067,6.477,148.907
C02724=1158.495,105.426,-53.630,-179.065,6.478,148.907
C02725=1158.490,105.694,-53.652,-179.062,6.479,148.906
C02726=1158.485,105.963,-53.671,-179.059,6.481,148.906
C02727=1158.479,106.231,-53.691,-179.056,6.483,148.905
C02728=1158.474,106.499,-53.711,-179.053,6.484,148.905
C02729=1158.470,106.749,-53.729,-179.050,6.486,148.904
C02730=1158.464,106.998,-53.748,-179.048,6.487,148.904
C02731=1158.460,107.247,-53.767,-179.044,6.489,148.903
C02732=1158.455,107.497,-53.786,-179.042,6.490,148.903
C02733=1158.450,107.746,-53.804,-179.040,6.491,148.902
C02734=1158.446,107.995,-53.823,-179.037,6.493,148.902
C02735=1158.440,108.244,-53.842,-179.034,6.495,148.902
C02736=1158.435,108.493,-53.860,-179.031,6.496,148.901
C02737=1158.431,108.743,-53.880,-179.028,6.498,148.901
C02738=1158.426,108.992,-53.898,-179.026,6.499,148.900
C02739=1158.421,109.241,-53.916,-179.023,6.500,148.900
C02740=1158.416,109.491,-53.935,-179.020,6.502,148.899
C02741=1158.411,109.739,-53.954,-179.017,6.503,148.899
C02742=1158.407,109.989,-53.974,-179.015,6.505,148.898
C02743=1158.402,110.238,-53.992,-179.012,6.507,148.898
C02744=1158.396,110.487,-54.011,-179.010,6.508,148.897
C02745=1158.392,110.737,-54.029,-179.007,6.509,148.897
C02746=1158.387,110.986,-54.048,-179.004,6.511,148.896
C02747=1158.383,111.235,-54.068,-179.001,6.513,148.896
C02748=1158.377,111.485,-54.086,-178.998,6.514,148.896
C02749=1158.373,111.733,-54.105,-178.996,6.515,148.895
C02750=1158.367,111.983,-54.124,-178.993,6.516,148.895
C02751=1158.363,112.232,-54.142,-178.990,6.518,148.894
C02752=1158.358,112.481,-54.162,-178.988,6.520,148.894
C02753=1158.353,112.731,-54.180,-178.985,6.522,148.893
C02754=1158.348,112.980,-54.200,-178.982,6.523,148.893
C02755=1158.344,113.229,-54.218,-178.980,6.524,148.892
C02756=1158.339,113.479,-54.237,-178.977,6.526,148.892
C02757=1158.333,113.728,-54.257,-178.974,6.527,148.892
C02758=1158.329,113.976,-54.275,-178.971,6.529,148.891
C02759=1158.324,114.226,-54.295,-178.969,6.531,148.891
C02760=1158.319,114.475,-54.313,-178.966,6.532,148.890
C02761=1158.314,114.725,-54.333,-178.963,6.534,148.890
C02762=1158.310,114.973,-54.351,-178.961,6.535,148.889
C02763=1158.305,115.223,-54.371,-178.958,6.536,148.889
C02764=1158.300,115.472,-54.390,-178.955,6.538,148.888
C02765=1158.295,115.722,-54.409,-178.953,6.540,148.888
C02766=1158.290,115.970,-54.428,-178.950,6.541,148.888
C02767=1158.285,116.220,-54.448,-178.947,6.543,148.887
C02768=1158.281,116.469,-54.466,-178.944,6.545,148.887
C02769=1158.276,116.718,-54.486,-178.942,6.545,148.886
C02770=1158.271,116.967,-54.505,-178.939,6.547,148.886
C02771=1158.266,117.217,-54.524,-178.936,6.549,148.885
C02772=1158.261,117.466,-54.543,-178.933,6.550,148.885
C02773=1158.256,117.715,-54.562,-178.930,6.552,148.884
C02774=1158.252,117.965,-54.582,-178.928,6.554,148.884
C02775=1158.247,118.213,-54.601,-178.925,6.555,148.884
C02776=1158.242,118.463,-54.620,-178.923,6.556,148.883
C02777=1158.238,118.712,-54.639,-178.920,6.558,148.883
C02778=1158.233,118.961,-54.659,-178.917,6.560,148.882
C02779=1158.228,119.210,-54.678,-178.914,6.561,148.882
C02780=1158.223,119.460,-54.698,-178.912,6.563,148.881
C02781=1158.219,119.709,-54.717,-178.909,6.564,148.881
C02782=1158.213,119.958,-54.736,-178.906,6.566,148.881
C02783=1158.209,120.207,-54.756,-178.903,6.568,148.880
C02784=1158.203,120.456,-54.775,-178.901,6.570,148.880
C02785=1158.199,120.705,-54.794,-178.898,6.570,148.879
C02786=1158.194,120.954,-54.813,-178.895,6.572,148.879
C02787=1158.189,121.204,-54.833,-178.893,6.574,148.878
C02788=1158.185,121.453,-54.853,-178.890,6.575,148.878
C02789=1158.180,121.702,-54.871,-178.887,6.577,148.877
C02790=1158.175,121.951,-54.891,-178.884,6.579,148.877
C02791=1158.170,122.201,-54.911,-178.882,6.580,148.877
C02792=1158.165,122.450,-54.930,-178.879,6.582,148.876
C02793=1158.160,122.700,-54.950,-178.876,6.583,148.876
C02794=1158.155,122.948,-54.969,-178.873,6.585,148.875
C02795=1158.151,123.197,-54.989,-178.871,6.586,148.875
C02796=1158.147,123.447,-55.008,-178.868,6.588,148.874
C02797=1158.141,123.695,-55.028,-178.866,6.589,148.874
C02798=1158.136,123.945,-55.047,-178.863,6.591,148.874
C02799=1158.132,124.195,-55.067,-178.860,6.593,148.873
C02800=1158.126,124.443,-55.086,-178.857,6.594,148.873
C02801=1158.122,124.692,-55.107,-178.854,6.596,148.872
C02802=1158.118,124.942,-55.126,-178.852,6.598,148.872
C02803=1158.113,125.191,-55.145,-178.849,6.599,148.871
C02804=1158.108,125.440,-55.165,-178.846,6.601,148.871
C02805=1158.103,125.690,-55.184,-178.843,6.603,148.871
C02806=1158.099,125.939,-55.205,-178.841,6.605,148.870
C02807=1158.093,126.187,-55.224,-178.838,6.606,148.870
C02808=1158.089,126.437,-55.244,-178.836,6.607,148.869
C02809=1158.084,126.687,-55.263,-178.833,6.609,148.869
C02810=1158.079,126.935,-55.283,-178.830,6.610,148.868
C02811=1158.074,127.184,-55.303,-178.827,6.612,148.868
C02812=1158.069,127.434,-55.323,-178.824,6.614,148.868
C02813=1158.065,127.683,-55.343,-178.822,6.615,148.867
C02814=1158.060,127.932,-55.362,-178.819,6.617,148.867
C02815=1158.055,128.181,-55.382,-178.816,6.619,148.866
C02816=1158.050,128.430,-55.402,-178.814,6.621,148.866
C02817=1158.046,128.680,-55.422,-178.811,6.622,148.866
C02818=1158.040,128.929,-55.441,-178.808,6.624,148.865
C02819=1158.036,129.178,-55.462,-178.805,6.625,148.865
C02820=1158.031,129.427,-55.481,-178.802,6.627,148.864
C02821=1158.027,129.676,-55.502,-178.800,6.629,148.864
C02822=1158.021,129.925,-55.521,-178.797,6.631,148.863
C02823=1158.017,130.174,-55.541,-178.794,6.632,148.863
C02824=1158.012,130.424,-55.561,-178.791,6.634,148.863
C02825=1158.007,130.673,-55.581,-178.789,6.636,148.862
C02826=1158.003,130.922,-55.601,-178.786,6.637,148.862
C02827=1157.998,131.171,-55.620,-178.783,6.639,148.861
C02828=1157.993,131.420,-55.641,-178.781,6.640,148.861
C02829=1157.987,131.689,-55.662,-178.777,6.642,148.860
C02830=1157.983,131.957,-55.684,-178.775,6.644,148.860
C02831=1157.977,132.226,-55.706,-178.772,6.646,148.860
C02832=1157.972,132.495,-55.727,-178.769,6.647,148.859
C02833=1157.968,132.743,-55.747,-178.767,6.649,148.859
C02834=1157.963,132.993,-55.767,-178.764,6.651,148.859
C02835=1157.959,133.242,-55.787,-178.761,6.652,148.858
C02836=1157.953,133.491,-55.807,-178.758,6.654,148.858
C02837=1157.948,133.740,-55.828,-178.755,6.656,148.857
C02838=1157.944,133.989,-55.848,-178.753,6.657,148.857
C02839=1157.939,134.239,-55.868,-178.750,6.659,148.856
C02840=1157.935,134.488,-55.888,-178.747,6.661,148.856
C02841=1157.930,134.737,-55.908,-178.744,6.662,148.856
C02842=1157.925,134.986,-55.929,-178.742,6.664,148.855
C02843=1157.920,135.235,-55.949,-178.739,6.666,148.855
C02844=1157.915,135.484,-55.968,-178.736,6.668,148.854
C02845=1157.910,135.733,-55.989,-178.734,6.669,148.854
C02846=1157.905,135.982,-56.010,-178.731,6.671,148.854
C02847=1157.901,136.231,-56.030,-178.728,6.673,148.853
C02848=1157.896,136.481,-56.050,-178.725,6.675,148.853
C02849=1157.892,136.730,-56.070,-178.723,6.676,148.852
C02850=1157.887,136.979,-56.090,-178.720,6.678,148.852
C02851=1157.882,137.229,-56.111,-178.717,6.680,148.852
C02852=1157.877,137.478,-56.131,-178.715,6.681,148.851
C02853=1157.872,137.726,-56.151,-178.712,6.683,148.851
C02854=1157.867,137.975,-56.172,-178.709,6.685,148.850
C02855=1157.863,138.224,-56.192,-178.706,6.686,148.850
C02856=1157.858,138.474,-56.212,-178.703,6.688,148.849
C02857=1157.853,138.723,-56.232,-178.701,6.690,148.849
C02858=1157.848,138.972,-56.253,-178.698,6.691,148.849
C02859=1157.844,139.221,-56.274,-178.695,6.693,148.848
C02860=1157.839,139.470,-56.294,-178.692,6.695,148.848
C02861=1157.834,139.719,-56.315,-178.690,6.697,148.848
C02862=1157.829,139.969,-56.335,-178.687,6.698,148.847
C02863=1157.825,140.218,-56.355,-178.684,6.701,148.847
C02864=1157.820,140.467,-56.376,-178.681,6.703,148.846
C02865=1157.815,140.716,-56.396,-178.678,6.704,148.846
C02866=1157.810,140.965,-56.417,-178.676,6.706,148.846
C02867=1157.806,141.214,-56.438,-178.673,6.708,148.845
C02868=1157.801,141.463,-56.458,-178.670,6.709,148.845
C02869=1157.796,141.712,-56.479,-178.668,6.711,148.844
C02870=1157.792,141.961,-56.499,-178.665,6.713,148.844
C02871=1157.787,142.210,-56.520,-178.662,6.715,148.844
C02872=1157.782,142.459,-56.541,-178.659,6.716,148.843
C02873=1157.778,142.708,-56.561,-178.657,6.718,148.843
C02874=1157.773,142.958,-56.582,-178.654,6.720,148.843
C02875=1157.768,143.207,-56.603,-178.651,6.722,148.842
C02876=1157.763,143.456,-56.624,-178.649,6.723,148.842
C02877=1157.759,143.705,-56.644,-178.646,6.725,148.841
C02878=1157.753,143.954,-56.665,-178.643,6.727,148.841
C02879=1157.749,144.203,-56.685,-178.640,6.728,148.841
C02880=1157.744,144.452,-56.706,-178.638,6.730,148.840
C02881=1157.739,144.701,-56.727,-178.635,6.732,148.840
C02882=1157.735,144.951,-56.747,-178.632,6.734,148.839
C02883=1157.730,145.200,-56.768,-178.629,6.736,148.839
C02884=1157.726,145.449,-56.789,-178.626,6.738,148.839
C02885=1157.721,145.698,-56.810,-178.624,6.740,148.838
C02886=1157.717,145.947,-56.831,-178.621,6.741,148.838
C02887=1157.711,146.196,-56.852,-178.618,6.743,148.838
C02888=1157.706,146.445,-56.873,-178.616,6.745,148.837
C02889=1157.702,146.694,-56.893,-178.613,6.747,148.837
C02890=1157.697,146.943,-56.914,-178.610,6.748,148.836
C02891=1157.692,147.192,-56.934,-178.607,6.750,148.836
C02892=1157.687,147.441,-56.956,-178.605,6.752,148.836
C02893=1157.683,147.691,-56.977,-178.602,6.753,148.835
C02894=1157.678,147.940,-56.998,-178.599,6.756,148.835
C02895=1157.673,148.189,-57.019,-178.596,6.758,148.834
C02896=1157.669,148.437,-57.040,-178.593,6.759,148.834
C02897=1157.664,148.687,-57.061,-178.591,6.762,148.834
C02898=1157.659,148.936,-57.081,-178.588,6.763,148.834
C02899=1157.654,149.185,-57.102,-178.586,6.765,148.833
C02900=1157.650,149.434,-57.124,-178.583,6.767,148.833
C02901=1157.645,149.683,-57.145,-178.580,6.768,148.832
C02902=1157.640,149.932,-57.165,-178.578,6.770,148.832
C02903=1157.635,150.181,-57.187,-178.575,6.772,148.832
C02904=1157.631,150.430,-57.208,-178.572,6.775,148.831
C02905=1157.626,150.679,-57.228,-178.569,6.776,148.831
C02906=1157.622,150.929,-57.251,-178.566,6.778,148.831
C02907=1157.617,151.178,-57.271,-178.564,6.780,148.830
C02908=1157.612,151.427,-57.292,-178.561,6.781,148.830
C02909=1157.607,151.675,-57.314,-178.558,6.783,148.829
C02910=1157.603,151.924,-57.334,-178.555,6.785,148.829
C02911=1157.598,152.173,-57.356,-178.553,6.787,148.829
C02912=1157.593,152.423,-57.377,-178.550,6.788,148.828
C02913=1157.588,152.672,-57.399,-178.547,6.791,148.828
C02914=1157.584,152.921,-57.419,-178.544,6.793,148.827
C02915=1157.579,153.170,-57.440,-178.541,6.794,148.827
C02916=1157.574,153.419,-57.462,-178.539,6.796,148.827
C02917=1157.569,153.668,-57.483,-178.536,6.798,148.827
C02918=1157.565,153.917,-57.504,-178.534,6.800,148.826
C02919=1157.560,154.166,-57.525,-178.531,6.802,148.826
C02920=1157.556,154.415,-57.547,-178.528,6.804,148.825
C02921=1157.550,154.665,-57.568,-178.525,6.806,148.825
C02922=1157.546,154.913,-57.590,-178.522,6.808,148.825
C02923=1157.541,155.162,-57.611,-178.520,6.809,148.824
C02924=1157.537,155.412,-57.632,-178.517,6.811,148.824
C02925=1157.532,155.660,-57.654,-178.514,6.813,148.824
C02926=1157.527,155.910,-57.675,-178.511,6.815,148.823
C02927=1157.522,156.158,-57.696,-178.508,6.817,148.823
C02928=1157.518,156.407,-57.719,-178.506,6.819,148.823
C02929=1157.513,156.657,-57.739,-178.503,6.821,148.822
C02930=1157.508,156.905,-57.761,-178.501,6.823,148.822
C02931=1157.504,157.155,-57.782,-178.498,6.824,148.822
C02932=1157.499,157.404,-57.804,-178.495,6.826,148.821
C02933=1157.494,157.673,-57.827,-178.492,6.829,148.821
C02934=1157.489,157.941,-57.850,-178.489,6.830,148.820
C02935=1157.484,158.211,-57.874,-178.486,6.833,148.820
C02936=1157.479,158.480,-57.897,-178.483,6.835,148.820
C02937=1157.474,158.729,-57.918,-178.481,6.837,148.819
C02938=1157.469,158.977,-57.940,-178.478,6.838,148.819
C02939=1157.465,159.227,-57.961,-178.475,6.841,148.819
C02940=1157.460,159.476,-57.983,-178.472,6.843,148.818
C02941=1157.455,159.724,-58.005,-178.469,6.844,148.818
C02942=1157.451,159.974,-58.027,-178.466,6.846,148.817
C02943=1157.446,160.222,-58.048,-178.464,6.848,148.817
C02944=1157.440,160.472,-58.069,-178.462,6.850,148.817
C02945=1157.436,160.721,-58.091,-178.458,6.852,148.817
C02946=1157.431,160.970,-58.113,-178.456,6.854,148.816
C02947=1157.427,161.219,-58.135,-178.453,6.856,148.816
C02948=1157.422,161.468,-58.157,-178.450,6.858,148.815
C02949=1157.417,161.716,-58.178,-178.447,6.859,148.815
C02950=1157.413,161.966,-58.200,-178.444,6.862,148.815
C02951=1157.408,162.215,-58.221,-178.442,6.864,148.815
C02952=1157.404,162.464,-58.244,-178.439,6.866,148.814
C02953=1157.399,162.713,-58.265,-178.437,6.867,148.814
C02954=1157.394,162.961,-58.287,-178.434,6.869,148.813
C02955=1157.390,163.211,-58.309,-178.431,6.872,148.813
C02956=1157.385,163.459,-58.331,-178.428,6.873,148.813
C02957=1157.380,163.709,-58.353,-178.425,6.875,148.812
C02958=1157.376,163.957,-58.374,-178.423,6.877,148.812
C02959=1157.371,164.207,-58.396,-178.420,6.879,148.812
C02960=1157.366,164.455,-58.418,-178.417,6.882,148.811
C02961=1157.362,164.705,-58.440,-178.414,6.883,148.811
C02962=1157.357,164.954,-58.462,-178.412,6.885,148.811
C02963=1157.352,165.203,-58.484,-178.409,6.887,148.810
C02964=1157.347,165.452,-58.506,-178.406,6.890,148.810
C02965=1157.343,165.701,-58.528,-178.403,6.891,148.810
C02966=1157.338,165.950,-58.550,-178.401,6.893,148.809
C02967=1157.333,166.198,-58.572,-178.398,6.895,148.809
C02968=1157.329,166.448,-58.594,-178.395,6.897,148.809
C02969=1157.324,166.697,-58.616,-178.392,6.899,148.808
C02970=1157.319,166.946,-58.638,-178.390,6.901,148.808
C02971=1157.314,167.195,-58.660,-178.387,6.903,148.808
C02972=1157.310,167.443,-58.682,-178.384,6.905,148.807
C02973=1157.306,167.692,-58.704,-178.381,6.907,148.807
C02974=1157.301,167.942,-58.727,-178.378,6.909,148.807
C02975=1157.296,168.191,-58.749,-178.376,6.911,148.806
C02976=1157.291,168.440,-58.770,-178.374,6.913,148.806
C02977=1157.287,168.689,-58.792,-178.370,6.916,148.806
C02978=1157.283,168.937,-58.815,-178.368,6.917,148.806
C02979=1157.278,169.187,-58.838,-178.365,6.919,148.805
C02980=1157.273,169.435,-58.859,-178.362,6.921,148.805
C02981=1157.268,169.685,-58.881,-178.359,6.924,148.805
C02982=1157.263,169.934,-58.904,-178.357,6.925,148.804
C02983=1157.259,170.182,-58.926,-178.354,6.927,148.804
C02984=1157.254,170.431,-58.948,-178.351,6.929,148.804
C02985=1157.250,170.680,-58.970,-178.348,6.931,148.803
C02986=1157.245,170.929,-58.993,-178.346,6.934,148.803
C02987=1157.240,171.178,-59.015,-178.343,6.935,148.803
C02988=1157.236,171.427,-59.037,-178.340,6.937,148.802
C02989=1157.230,171.676,-59.059,-178.337,6.940,148.802
C02990=1157.226,171.925,-59.082,-178.334,6.941,148.802
C02991=1157.222,172.174,-59.104,-178.332,6.943,148.801
C02992=1157.216,172.423,-59.126,-178.329,6.946,148.801
C02993=1157.213,172.672,-59.149,-178.326,6.948,148.801
C02994=1157.208,172.921,-59.171,-178.324,6.950,148.800
C02995=1157.203,173.170,-59.194,-178.321,6.952,148.800
C02996=1157.199,173.419,-59.216,-178.318,6.954,148.800
C02997=1157.193,173.668,-59.239,-178.315,6.956,148.799
C02998=1157.189,173.917,-59.261,-178.313,6.958,148.799
C02999=1157.185,174.166,-59.283,-178.310,6.959,148.799
C03000=1157.180,174.414,-59.306,-178.307,6.962,148.799
C03001=1157.175,174.664,-59.328,-178.305,6.964,148.798
C03002=1157.171,174.913,-59.352,-178.302,6.966,148.798
C03003=1157.166,175.161,-59.374,-178.299,6.968,148.798
C03004=1157.161,175.410,-59.397,-178.296,6.970,148.797
C03005=1157.157,175.660,-59.419,-178.294,6.972,148.797
C03006=1157.151,175.908,-59.442,-178.290,6.975,148.797
C03007=1157.147,176.157,-59.464,-178.288,6.977,148.796
C03008=1157.143,176.406,-59.487,-178.285,6.979,148.796
C03009=1157.138,176.655,-59.509,-178.283,6.980,148.796
C03010=1157.134,176.904,-59.532,-178.280,6.983,148.795
C03011=1157.129,177.153,-59.555,-178.277,6.985,148.795
C03012=1157.124,177.401,-59.577,-178.275,6.987,148.795
C03013=1157.119,177.650,-59.600,-178.271,6.989,148.795
C03014=1157.115,177.900,-59.622,-178.269,6.991,148.794
C03015=1157.110,178.149,-59.646,-178.266,6.993,148.794
C03016=1157.105,178.397,-59.669,-178.263,6.996,148.794
C03017=1157.101,178.646,-59.691,-178.260,6.997,148.793
C03018=1157.096,178.896,-59.714,-178.258,6.999,148.793
C03019=1157.092,179.144,-59.737,-178.255,7.002,148.793
C03020=1157.087,179.393,-59.759,-178.252,7.004,148.793
C03021=1157.083,179.642,-59.782,-178.250,7.006,148.792
C03022=1157.078,179.891,-59.805,-178.246,7.008,148.792
C03023=1157.073,180.140,-59.828,-178.244,7.010,148.792
C03024=1157.068,180.389,-59.850,-178.241,7.012,148.791
C03025=1157.064,180.638,-59.874,-178.238,7.015,148.791
C03026=1157.060,180.886,-59.896,-178.236,7.017,148.791
C03027=1157.055,181.135,-59.920,-178.233,7.018,148.791
C03028=1157.050,181.385,-59.942,-178.230,7.021,148.790
C03029=1157.045,181.633,-59.965,-178.227,7.023,148.790
C03030=1157.041,181.882,-59.988,-178.225,7.025,148.790
C03031=1157.036,182.131,-60.011,-178.222,7.027,148.789
C03032=1157.032,182.380,-60.034,-178.219,7.029,148.789
C03033=1157.027,182.629,-60.058,-178.217,7.031,148.789
C03034=1157.022,182.878,-60.080,-178.214,7.034,148.788
C03035=1157.018,183.127,-60.103,-178.211,7.036,148.788
C03036=1157.013,183.376,-60.126,-178.208,7.037,148.788
C03037=1157.008,183.645,-60.151,-178.205,7.040,148.788
C03038=1157.003,183.915,-60.175,-178.202,7.043,148.787
C03039=1156.998,184.184,-60.201,-178.200,7.045,148.787
C03040=1156.993,184.454,-60.226,-178.196,7.047,148.787
C03041=1156.989,184.702,-60.249,-178.194,7.049,148.786
C03042=1156.984,184.951,-60.272,-178.191,7.052,148.786
C03043=1156.980,185.201,-60.296,-178.188,7.054,148.786
C03044=1156.975,185.450,-60.319,-178.185,7.055,148.785
C03045=1156.970,185.699,-60.342,-178.183,7.058,148.785
C03046=1156.966,185.947,-60.365,-178.180,7.060,148.785
C03047=1156.961,186.196,-60.389,-178.177,7.063,148.785
C03048=1156.956,186.445,-60.412,-178.174,7.065,148.784
C03049=1156.951,186.694,-60.435,-178.172,7.066,148.784
C03050=1156.947,186.943,-60.458,-178.168,7.069,148.784
C03051=1156.943,187.191,-60.481,-178.166,7.071,148.784
C03052=1156.938,187.440,-60.504,-178.163,7.074,148.783
C03053=1156.933,187.690,-60.528,-178.160,7.075,148.783
C03054=1156.929,187.939,-60.551,-178.158,7.078,148.783
C03055=1156.924,188.188,-60.574,-178.155,7.080,148.782
C03056=1156.919,188.437,-60.598,-178.153,7.082,148.782
C03057=1156.916,188.685,-60.621,-178.150,7.084,148.782
C03058=1156.911,188.934,-60.645,-178.147,7.087,148.782
C03059=1156.906,189.183,-60.668,-178.144,7.089,148.782
C03060=1156.902,189.432,-60.691,-178.141,7.091,148.781
C03061=1156.896,189.680,-60.714,-178.139,7.093,148.781
C03062=1156.892,189.929,-60.738,-178.136,7.095,148.781
C03063=1156.887,190.178,-60.762,-178.133,7.098,148.780
C03064=1156.882,190.427,-60.785,-178.130,7.099,148.780
C03065=1156.878,190.676,-60.808,-178.128,7.102,148.780
C03066=1156.873,190.925,-60.832,-178.125,7.104,148.780
C03067=1156.869,191.173,-60.856,-178.122,7.107,148.779
C03068=1156.864,191.422,-60.879,-178.119,7.109,148.779
C03069=1156.859,191.671,-60.903,-178.117,7.110,148.779
C03070=1156.855,191.920,-60.926,-178.114,7.113,148.779
C03071=1156.850,192.169,-60.950,-178.111,7.115,148.778
C03072=1156.845,192.418,-60.973,-178.108,7.118,148.778
C03073=1156.841,192.667,-60.997,-178.106,7.120,148.778
C03074=1156.836,192.915,-61.021,-178.103,7.122,148.777
C03075=1156.832,193.164,-61.044,-178.100,7.125,148.777
C03076=1156.827,193.413,-61.068,-178.098,7.126,148.777
C03077=1156.823,193.662,-61.092,-178.094,7.129,148.777
C03078=1156.818,193.911,-61.115,-178.092,7.131,148.776
C03079=1156.814,194.160,-61.139,-178.089,7.134,148.776
C03080=1156.809,194.409,-61.163,-178.087,7.136,148.776
C03081=1156.805,194.657,-61.187,-178.083,7.138,148.776
C03082=1156.800,194.906,-61.210,-178.081,7.140,148.775
C03083=1156.796,195.155,-61.234,-178.079,7.142,148.775
C03084=1156.791,195.404,-61.258,-178.075,7.145,148.775
C03085=1156.786,195.653,-61.281,-178.073,7.147,148.775
C03086=1156.782,195.901,-61.305,-178.070,7.149,148.774
C03087=1156.777,196.150,-61.329,-178.067,7.151,148.774
C03088=1156.772,196.399,-61.353,-178.064,7.154,148.774
C03089=1156.768,196.648,-61.377,-178.062,7.156,148.774
C03090=1156.764,196.897,-61.401,-178.059,7.159,148.774
C03091=1156.759,197.145,-61.425,-178.056,7.160,148.773
C03092=1156.755,197.394,-61.448,-178.053,7.163,148.773
C03093=1156.750,197.643,-61.472,-178.051,7.165,148.773
C03094=1156.745,197.892,-61.496,-178.048,7.167,148.772
C03095=1156.740,198.141,-61.520,-178.045,7.170,148.772
C03096=1156.736,198.390,-61.544,-178.043,7.172,148.772
C03097=1156.731,198.638,-61.568,-178.040,7.174,148.772
C03098=1156.728,198.887,-61.592,-178.037,7.176,148.771
C03099=1156.722,199.136,-61.616,-178.034,7.179,148.771
C03100=1156.718,199.385,-61.640,-178.032,7.181,148.771
C03101=1156.713,199.633,-61.664,-178.029,7.184,148.771
C03102=1156.709,199.882,-61.688,-178.026,7.186,148.771
C03103=1156.704,200.131,-61.712,-178.023,7.188,148.770
C03104=1156.700,200.380,-61.737,-178.021,7.190,148.770
C03105=1156.695,200.629,-61.761,-178.017,7.193,148.770
C03106=1156.691,200.878,-61.784,-178.015,7.195,148.770
C03107=1156.685,201.126,-61.809,-178.012,7.198,148.769
C03108=1156.681,201.375,-61.833,-178.010,7.200,148.769
C03109=1156.677,201.624,-61.858,-178.006,7.202,148.769
C03110=1156.673,201.873,-61.881,-178.004,7.204,148.769
C03111=1156.667,202.122,-61.906,-178.001,7.207,148.768
C03112=1156.663,202.370,-61.930,-177.999,7.209,148.768
C03113=1156.659,202.619,-61.954,-177.996,7.212,148.768
C03114=1156.654,202.868,-61.979,-177.993,7.214,148.768
C03115=1156.650,203.116,-62.003,-177.990,7.216,148.767
C03116=1156.645,203.365,-62.026,-177.988,7.218,148.767
C03117=1156.640,203.614,-62.051,-177.985,7.221,148.767
C03118=1156.636,203.863,-62.075,-177.982,7.223,148.767
C03119=1156.632,204.112,-62.099,-177.979,7.226,148.767
C03120=1156.627,204.360,-62.124,-177.977,7.228,148.766
C03121=1156.623,204.609,-62.148,-177.974,7.230,148.766
C03122=1156.618,204.858,-62.173,-177.971,7.232,148.766
C03123=1156.613,205.107,-62.197,-177.968,7.235,148.766
C03124=1156.609,205.355,-62.221,-177.966,7.237,148.766
C03125=1156.604,205.604,-62.246,-177.963,7.240,148.765
C03126=1156.600,205.853,-62.270,-177.961,7.242,148.765
C03127=1156.595,206.102,-62.295,-177.957,7.244,148.765
C03128=1156.591,206.351,-62.320,-177.955,7.247,148.765
C03129=1156.586,206.599,-62.344,-177.952,7.249,148.764
C03130=1156.582,206.848,-62.368,-177.950,7.251,148.764
C03131=1156.576,207.096,-62.393,-177.946,7.254,148.764
C03132=1156.573,207.346,-62.417,-177.944,7.257,148.764
C03133=1156.567,207.594,-62.442,-177.941,7.258,148.763
C03134=1156.563,207.843,-62.466,-177.938,7.261,148.763
C03135=1156.559,208.092,-62.491,-177.935,7.263,148.763
C03136=1156.554,208.341,-62.515,-177.933,7.266,148.763
C03137=1156.549,208.589,-62.540,-177.930,7.268,148.763
C03138=1156.545,208.838,-62.564,-177.927,7.271,148.762
C03139=1156.540,209.087,-62.590,-177.924,7.273,148.762
C03140=1156.537,209.336,-62.614,-177.922,7.275,148.762
C03141=1156.531,209.606,-62.641,-177.918,7.278,148.762
C03142=1156.526,209.876,-62.668,-177.916,7.281,148.762
C03143=1156.522,210.147,-62.695,-177.913,7.283,148.761
C03144=1156.516,210.417,-62.722,-177.910,7.286,148.761
C03145=1156.512,210.666,-62.746,-177.907,7.288,148.761
C03146=1156.507,210.915,-62.771,-177.905,7.290,148.761
C03147=1156.503,211.164,-62.795,-177.901,7.293,148.760
C03148=1156.498,211.413,-62.820,-177.899,7.296,148.760
C03149=1156.493,211.661,-62.846,-177.896,7.298,148.760
C03150=1156.489,211.910,-62.870,-177.893,7.301,148.760
C03151=1156.484,212.159,-62.895,-177.891,7.302,148.760
C03152=1156.480,212.408,-62.920,-177.888,7.305,148.759
C03153=1156.476,212.656,-62.945,-177.886,7.307,148.759
C03154=1156.470,212.905,-62.969,-177.882,7.310,148.759
C03155=1156.466,213.154,-62.995,-177.880,7.313,148.759
C03156=1156.462,213.402,-63.019,-177.877,7.315,148.759
C03157=1156.457,213.652,-63.044,-177.874,7.318,148.758
C03158=1156.453,213.900,-63.069,-177.871,7.319,148.758
C03159=1156.449,214.149,-63.094,-177.869,7.322,148.758
C03160=1156.444,214.397,-63.119,-177.866,7.325,148.758
C03161=1156.439,214.646,-63.144,-177.863,7.327,148.758
C03162=1156.434,214.895,-63.169,-177.860,7.330,148.758
C03163=1156.431,215.143,-63.194,-177.858,7.332,148.757
C03164=1156.426,215.392,-63.219,-177.855,7.335,148.757
C03165=1156.421,215.641,-63.245,-177.852,7.338,148.757
C03166=1156.416,215.890,-63.269,-177.849,7.339,148.757
C03167=1156.413,216.138,-63.294,-177.847,7.342,148.757
C03168=1156.408,216.387,-63.319,-177.844,7.344,148.756
C03169=1156.403,216.636,-63.345,-177.841,7.347,148.756
C03170=1156.398,216.884,-63.369,-177.838,7.350,148.756
C03171=1156.395,217.133,-63.395,-177.836,7.352,148.756
C03172=1156.390,217.381,-63.420,-177.833,7.355,148.756
C03173=1156.385,217.631,-63.445,-177.830,7.356,148.755
C03174=1156.381,217.879,-63.470,-177.828,7.359,148.755
C03175=1156.376,218.128,-63.495,-177.825,7.362,148.755
C03176=1156.372,218.377,-63.521,-177.822,7.364,148.755
C03177=1156.368,218.625,-63.546,-177.819,7.367,148.755
C03178=1156.363,218.874,-63.571,-177.816,7.370,148.755
C03179=1156.358,219.122,-63.596,-177.814,7.372,148.754
C03180=1156.354,219.371,-63.622,-177.811,7.375,148.754
C03181=1156.349,219.620,-63.647,-177.808,7.376,148.754
C03182=1156.345,219.868,-63.673,-177.806,7.379,148.754
C03183=1156.341,220.117,-63.698,-177.803,7.382,148.754
C03184=1156.335,220.366,-63.723,-177.800,7.384,148.753
C03185=1156.331,220.615,-63.749,-177.797,7.387,148.753
C03186=1156.326,220.863,-63.774,-177.795,7.390,148.753
C03187=1156.323,221.111,-63.799,-177.792,7.392,148.753
C03188=1156.318,221.361,-63.824,-177.789,7.394,148.753
C03189=1156.314,221.609,-63.850,-177.786,7.397,148.753
C03190=1156.309,221.858,-63.875,-177.784,7.399,148.752
C03191=1156.305,222.107,-63.901,-177.781,7.402,148.752
C03192=1156.300,222.355,-63.927,-177.778,7.405,148.752
C03193=1156.296,222.604,-63.952,-177.775,7.407,148.752
C03194=1156.291,222.852,-63.977,-177.773,7.410,148.752
C03195=1156.287,223.101,-64.003,-177.770,7.412,148.752
C03196=1156.282,223.350,-64.029,-177.767,7.414,148.751
C03197=1156.278,223.598,-64.054,-177.764,7.417,148.751
C03198=1156.273,223.847,-64.080,-177.762,7.419,148.751
C03199=1156.269,224.096,-64.105,-177.759,7.422,148.751
C03200=1156.264,224.344,-64.131,-177.756,7.425,148.751
C03201=1156.259,224.593,-64.157,-177.754,7.427,148.751
C03202=1156.255,224.842,-64.182,-177.751,7.430,148.750
C03203=1156.250,225.090,-64.208,-177.748,7.433,148.750
C03204=1156.246,225.339,-64.233,-177.745,7.436,148.750
C03205=1156.242,225.588,-64.259,-177.742,7.437,148.750
C03206=1156.237,225.837,-64.285,-177.740,7.440,148.750
C03207=1156.233,226.085,-64.310,-177.737,7.443,148.750
C03208=1156.228,226.334,-64.336,-177.734,7.445,148.749
C03209=1156.224,226.582,-64.362,-177.731,7.448,148.749
C03210=1156.219,226.832,-64.388,-177.729,7.451,148.749
C03211=1156.215,227.079,-64.414,-177.726,7.453,148.749
C03212=1156.210,227.328,-64.440,-177.723,7.456,148.749
C03213=1156.206,227.577,-64.466,-177.720,7.458,148.749
C03214=1156.201,227.825,-64.491,-177.718,7.461,148.748
C03215=1156.197,228.074,-64.517,-177.715,7.463,148.748
C03216=1156.192,228.323,-64.543,-177.712,7.466,148.748
C03217=1156.188,228.571,-64.569,-177.709,7.469,148.748
C03218=1156.184,228.820,-64.595,-177.707,7.471,148.748
C03219=1156.179,229.068,-64.620,-177.704,7.474,148.748
C03220=1156.175,229.317,-64.646,-177.701,7.477,148.747
C03221=1156.170,229.566,-64.673,-177.699,7.479,148.747
C03222=1156.166,229.814,-64.699,-177.696,7.481,148.747
C03223=1156.162,230.063,-64.724,-177.693,7.484,148.747
C03224=1156.157,230.311,-64.750,-177.690,7.487,148.747
C03225=1156.152,230.560,-64.777,-177.688,7.489,148.747
C03226=1156.148,230.809,-64.803,-177.685,7.492,148.746
C03227=1156.144,231.057,-64.828,-177.682,7.495,148.746
C03228=1156.140,231.306,-64.855,-177.680,7.497,148.746
C03229=1156.134,231.554,-64.881,-177.677,7.500,148.746
C03230=1156.130,231.803,-64.906,-177.674,7.503,148.746
C03231=1156.126,232.052,-64.932,-177.671,7.506,148.746
C03232=1156.121,232.300,-64.959,-177.669,7.508,148.746
C03233=1156.117,232.549,-64.985,-177.666,7.510,148.745
C03234=1156.113,232.798,-65.011,-177.663,7.513,148.745
C03235=1156.108,233.046,-65.038,-177.660,7.516,148.745
C03236=1156.103,233.294,-65.063,-177.658,7.518,148.745
C03237=1156.099,233.543,-65.090,-177.655,7.521,148.745
C03238=1156.094,233.792,-65.116,-177.652,7.524,148.745
C03239=1156.090,234.040,-65.142,-177.649,7.527,148.745
C03240=1156.085,234.289,-65.169,-177.647,7.529,148.745
C03241=1156.081,234.538,-65.195,-177.644,7.532,148.744
C03242=1156.077,234.786,-65.221,-177.641,7.534,148.744
C03243=1156.072,235.035,-65.247,-177.638,7.537,148.744
C03244=1156.068,235.283,-65.274,-177.636,7.539,148.744
C03245=1156.063,235.555,-65.303,-177.633,7.542,148.744
C03246=1156.059,235.827,-65.331,-177.630,7.545,148.744
C03247=1156.053,236.098,-65.361,-177.626,7.549,148.744
C03248=1156.049,236.370,-65.389,-177.624,7.552,148.743
C03249=1156.044,236.619,-65.416,-177.621,7.553,148.743
C03250=1156.040,236.868,-65.441,-177.618,7.556,148.743
C03251=1156.035,237.116,-65.469,-177.615,7.559,148.743
C03252=1156.031,237.364,-65.495,-177.613,7.562,148.743
C03253=1156.026,237.613,-65.521,-177.610,7.565,148.743
C03254=1156.022,237.862,-65.548,-177.607,7.567,148.743
C03255=1156.017,238.111,-65.574,-177.604,7.570,148.742
C03256=1156.013,238.358,-65.600,-177.602,7.573,148.742
C03257=1156.008,238.607,-65.627,-177.599,7.576,148.742
C03258=1156.004,238.855,-65.653,-177.597,7.578,148.742
C03259=1155.999,239.104,-65.680,-177.594,7.581,148.742
C03260=1155.995,239.352,-65.707,-177.591,7.583,148.742
C03261=1155.990,239.601,-65.733,-177.588,7.586,148.742
C03262=1155.986,239.850,-65.760,-177.585,7.589,148.742
C03263=1155.982,240.098,-65.786,-177.583,7.591,148.742
C03264=1155.977,240.346,-65.814,-177.580,7.594,148.741
C03265=1155.973,240.596,-65.840,-177.577,7.597,148.741
C03266=1155.969,240.844,-65.867,-177.574,7.600,148.741
C03267=1155.964,241.093,-65.894,-177.571,7.603,148.741
C03268=1155.960,241.341,-65.920,-177.569,7.605,148.741
C03269=1155.956,241.590,-65.947,-177.566,7.608,148.741
C03270=1155.951,241.839,-65.974,-177.564,7.611,148.741
C03271=1155.947,242.087,-66.000,-177.561,7.614,148.741
C03272=1155.942,242.335,-66.027,-177.558,7.616,148.740
C03273=1155.938,242.584,-66.054,-177.555,7.618,148.740
C03274=1155.934,242.832,-66.081,-177.553,7.621,148.740
C03275=1155.929,243.081,-66.108,-177.550,7.624,148.740
C03276=1155.924,243.329,-66.135,-177.547,7.627,148.740
C03277=1155.920,243.577,-66.161,-177.544,7.630,148.740
C03278=1155.916,243.826,-66.188,-177.542,7.632,148.740
C03279=1155.911,244.074,-66.215,-177.539,7.635,148.740
C03280=1155.906,244.323,-66.242,-177.536,7.638,148.740
C03281=1155.903,244.572,-66.269,-177.533,7.641,148.739
C03282=1155.898,244.821,-66.296,-177.531,7.644,148.739
C03283=1155.893,245.069,-66.323,-177.528,7.646,148.739
C03284=1155.889,245.318,-66.350,-177.526,7.649,148.739
C03285=1155.885,245.566,-66.376,-177.523,7.652,148.739
C03286=1155.881,245.814,-66.404,-177.520,7.655,148.739
C03287=1155.876,246.062,-66.431,-177.517,7.657,148.739
C03288=1155.872,246.311,-66.459,-177.514,7.660,148.739
C03289=1155.867,246.560,-66.486,-177.512,7.662,148.739
C03290=1155.863,246.808,-66.512,-177.509,7.665,148.739
C03291=1155.859,247.057,-66.539,-177.506,7.668,148.739
C03292=1155.854,247.305,-66.566,-177.503,7.671,148.738
C03293=1155.849,247.554,-66.593,-177.501,7.674,148.738
C03294=1155.845,247.802,-66.620,-177.498,7.677,148.738
C03295=1155.841,248.051,-66.648,-177.495,7.680,148.738
C03296=1155.836,248.299,-66.675,-177.493,7.682,148.738
C03297=1155.832,248.547,-66.702,-177.490,7.685,148.738
C03298=1155.828,248.796,-66.729,-177.487,7.688,148.738
C03299=1155.823,249.044,-66.756,-177.484,7.691,148.738
C03300=1155.819,249.294,-66.784,-177.481,7.693,148.738
C03301=1155.815,249.541,-66.811,-177.479,7.696,148.738
C03302=1155.810,249.790,-66.838,-177.476,7.699,148.737
C03303=1155.805,250.038,-66.865,-177.474,7.701,148.737
C03304=1155.801,250.288,-66.893,-177.471,7.704,148.737
C03305=1155.797,250.536,-66.921,-177.468,7.707,148.737
C03306=1155.792,250.784,-66.948,-177.465,7.710,148.737
C03307=1155.788,251.033,-66.975,-177.463,7.713,148.737
C03308=1155.784,251.281,-67.003,-177.460,7.716,148.737
C03309=1155.779,251.530,-67.030,-177.458,7.718,148.737
C03310=1155.774,251.778,-67.057,-177.455,7.721,148.737
C03311=1155.770,252.026,-67.085,-177.452,7.724,148.737
C03312=1155.766,252.275,-67.112,-177.449,7.727,148.737
C03313=1155.762,252.523,-67.140,-177.446,7.730,148.737
C03314=1155.757,252.772,-67.167,-177.444,7.733,148.737
C03315=1155.752,253.020,-67.194,-177.440,7.736,148.736
C03316=1155.749,253.269,-67.222,-177.438,7.739,148.736
C03317=1155.744,253.517,-67.249,-177.436,7.741,148.736
C03318=1155.740,253.765,-67.277,-177.433,7.744,148.736
C03319=1155.736,254.014,-67.305,-177.430,7.747,148.736
C03320=1155.731,254.262,-67.332,-177.427,7.750,148.736
C03321=1155.727,254.511,-67.359,-177.424,7.752,148.736
C03322=1155.723,254.759,-67.387,-177.422,7.755,148.736
C03323=1155.718,255.008,-67.415,-177.419,7.758,148.736
C03324=1155.714,255.255,-67.442,-177.416,7.761,148.736
C03325=1155.709,255.505,-67.470,-177.413,7.764,148.736
C03326=1155.705,255.753,-67.498,-177.411,7.766,148.736
C03327=1155.700,256.001,-67.526,-177.408,7.769,148.736
C03328=1155.696,256.250,-67.553,-177.406,7.772,148.735
C03329=1155.692,256.498,-67.581,-177.403,7.775,148.735
C03330=1155.687,256.746,-67.608,-177.400,7.778,148.735
C03331=1155.683,256.995,-67.637,-177.397,7.781,148.735
C03332=1155.678,257.243,-67.665,-177.394,7.784,148.735
C03333=1155.674,257.492,-67.692,-177.392,7.787,148.735
C03334=1155.670,257.740,-67.720,-177.389,7.790,148.735
C03335=1155.666,257.988,-67.748,-177.386,7.793,148.735
C03336=1155.661,258.238,-67.776,-177.383,7.796,148.735
C03337=1155.657,258.485,-67.803,-177.381,7.798,148.735
C03338=1155.653,258.734,-67.832,-177.378,7.801,148.735
C03339=1155.648,258.982,-67.859,-177.376,7.804,148.735
C03340=1155.643,259.231,-67.887,-177.373,7.807,148.735
C03341=1155.639,259.479,-67.915,-177.371,7.810,148.735
C03342=1155.635,259.727,-67.943,-177.368,7.813,148.735
C03343=1155.631,259.976,-67.971,-177.365,7.816,148.735
C03344=1155.626,260.224,-67.999,-177.362,7.819,148.735
C03345=1155.622,260.473,-68.027,-177.360,7.822,148.735
C03346=1155.618,260.721,-68.055,-177.357,7.825,148.735
C03347=1155.613,260.969,-68.083,-177.354,7.828,148.734
C03348=1155.609,261.218,-68.111,-177.351,7.831,148.734
C03349=1155.604,261.491,-68.142,-177.348,7.834,148.734
C03350=1155.600,261.764,-68.173,-177.346,7.836,148.734
C03351=1155.595,262.038,-68.203,-177.342,7.840,148.734
C03352=1155.589,262.311,-68.235,-177.340,7.843,148.734
C03353=1155.585,262.559,-68.262,-177.337,7.846,148.734
C03354=1155.581,262.808,-68.290,-177.334,7.849,148.734
C03355=1155.576,263.056,-68.319,-177.331,7.852,148.734
C03356=1155.573,263.305,-68.347,-177.328,7.855,148.734
C03357=1155.567,263.553,-68.375,-177.326,7.858,148.734
C03358=1155.564,263.801,-68.403,-177.323,7.861,148.734
C03359=1155.559,264.049,-68.431,-177.321,7.863,148.734
C03360=1155.555,264.298,-68.460,-177.318,7.866,148.734
C03361=1155.550,264.546,-68.488,-177.315,7.869,148.734
C03362=1155.546,264.795,-68.516,-177.313,7.872,148.734
C03363=1155.542,265.043,-68.545,-177.310,7.875,148.734
C03364=1155.537,265.291,-68.574,-177.307,7.878,148.734
C03365=1155.534,265.540,-68.602,-177.305,7.881,148.734
C03366=1155.529,265.788,-68.630,-177.302,7.884,148.734
C03367=1155.525,266.036,-68.658,-177.299,7.887,148.734
C03368=1155.520,266.285,-68.687,-177.296,7.890,148.733
C03369=1155.516,266.533,-68.715,-177.293,7.893,148.733
C03370=1155.511,266.781,-68.743,-177.291,7.896,148.733
C03371=1155.507,267.030,-68.771,-177.288,7.899,148.734
C03372=1155.503,267.278,-68.801,-177.286,7.902,148.733
C03373=1155.499,267.526,-68.829,-177.283,7.905,148.733
C03374=1155.494,267.775,-68.857,-177.280,7.908,148.733
C03375=1155.490,268.023,-68.885,-177.277,7.911,148.733
C03376=1155.486,268.271,-68.915,-177.275,7.914,148.733
C03377=1155.481,268.520,-68.943,-177.272,7.917,148.733
C03378=1155.477,268.768,-68.971,-177.269,7.920,148.733
C03379=1155.472,269.017,-69.000,-177.267,7.923,148.733
C03380=1155.469,269.265,-69.029,-177.264,7.926,148.733
C03381=1155.464,269.513,-69.057,-177.261,7.929,148.733
C03382=1155.459,269.762,-69.086,-177.258,7.932,148.733
C03383=1155.456,270.010,-69.115,-177.256,7.935,148.733
C03384=1155.451,270.258,-69.143,-177.253,7.938,148.733
C03385=1155.446,270.507,-69.172,-177.251,7.941,148.733
C03386=1155.442,270.754,-69.200,-177.248,7.944,148.733
C03387=1155.438,271.003,-69.229,-177.245,7.947,148.733
C03388=1155.434,271.251,-69.258,-177.242,7.950,148.733
C03389=1155.430,271.500,-69.287,-177.239,7.953,148.733
C03390=1155.425,271.748,-69.315,-177.237,7.956,148.733
C03391=1155.421,271.996,-69.344,-177.234,7.959,148.733
C03392=1155.417,272.245,-69.373,-177.232,7.962,148.733
C03393=1155.412,272.492,-69.402,-177.229,7.965,148.733
C03394=1155.408,272.741,-69.430,-177.226,7.968,148.733
C03395=1155.403,272.989,-69.460,-177.223,7.971,148.733
C03396=1155.399,273.237,-69.488,-177.221,7.974,148.733
C03397=1155.395,273.486,-69.517,-177.218,7.977,148.733
C03398=1155.390,273.735,-69.546,-177.215,7.980,148.733
C03399=1155.386,273.983,-69.575,-177.213,7.983,148.733
C03400=1155.382,274.231,-69.603,-177.210,7.986,148.733
C03401=1155.378,274.479,-69.633,-177.208,7.989,148.733
C03402=1155.373,274.727,-69.662,-177.205,7.992,148.733
C03403=1155.369,274.976,-69.691,-177.202,7.995,148.733
C03404=1155.365,275.223,-69.719,-177.199,7.998,148.733
C03405=1155.360,275.472,-69.748,-177.197,8.001,148.733
C03406=1155.356,275.720,-69.777,-177.194,8.004,148.733
C03407=1155.352,275.969,-69.807,-177.191,8.007,148.733
C03408=1155.348,276.218,-69.836,-177.189,8.010,148.733
C03409=1155.343,276.465,-69.865,-177.186,8.013,148.733
C03410=1155.339,276.713,-69.894,-177.184,8.016,148.733
C03411=1155.335,276.961,-69.923,-177.181,8.019,148.733
C03412=1155.331,277.210,-69.952,-177.178,8.022,148.733
C03413=1155.326,277.459,-69.981,-177.175,8.025,148.733
C03414=1155.322,277.706,-70.010,-177.173,8.028,148.733
C03415=1155.318,277.954,-70.040,-177.170,8.031,148.733
C03416=1155.313,278.203,-70.068,-177.167,8.034,148.733
C03417=1155.309,278.452,-70.098,-177.165,8.037,148.733
C03418=1155.305,278.700,-70.127,-177.162,8.040,148.733
C03419=1155.300,278.948,-70.157,-177.160,8.043,148.733
C03420=1155.296,279.196,-70.186,-177.157,8.046,148.733
C03421=1155.292,279.444,-70.215,-177.154,8.049,148.733
C03422=1155.288,279.693,-70.243,-177.152,8.053,148.733
C03423=1155.284,279.941,-70.273,-177.149,8.055,148.733
C03424=1155.279,280.189,-70.302,-177.146,8.058,148.733
C03425=1155.275,280.437,-70.332,-177.143,8.061,148.733
C03426=1155.271,280.686,-70.361,-177.141,8.065,148.733
C03427=1155.267,280.934,-70.391,-177.138,8.068,148.733
C03428=1155.263,281.182,-70.420,-177.136,8.071,148.733
C03429=1155.257,281.430,-70.450,-177.133,8.074,148.733
C03430=1155.253,281.678,-70.479,-177.130,8.078,148.733
C03431=1155.249,281.927,-70.509,-177.127,8.081,148.733
C03432=1155.245,282.175,-70.538,-177.124,8.084,148.733
C03433=1155.240,282.423,-70.568,-177.122,8.087,148.733
C03434=1155.236,282.671,-70.597,-177.119,8.090,148.733
C03435=1155.232,282.920,-70.627,-177.117,8.093,148.733
C03436=1155.228,283.168,-70.656,-177.114,8.096,148.733
C03437=1155.224,283.416,-70.686,-177.112,8.099,148.733
C03438=1155.220,283.664,-70.715,-177.109,8.102,148.733
C03439=1155.215,283.913,-70.744,-177.106,8.105,148.733
C03440=1155.210,284.161,-70.774,-177.104,8.108,148.733
C03441=1155.206,284.410,-70.804,-177.101,8.111,148.733
C03442=1155.202,284.657,-70.834,-177.099,8.114,148.733
C03443=1155.198,284.905,-70.863,-177.096,8.117,148.733
C03444=1155.193,285.153,-70.893,-177.093,8.120,148.733
C03445=1155.189,285.401,-70.922,-177.091,8.123,148.734
C03446=1155.185,285.650,-70.952,-177.087,8.127,148.734
C03447=1155.180,285.898,-70.982,-177.085,8.130,148.734
C03448=1155.176,286.146,-71.012,-177.082,8.133,148.734
C03449=1155.172,286.394,-71.041,-177.080,8.136,148.734
C03450=1155.168,286.642,-71.071,-177.077,8.139,148.734
C03451=1155.163,286.891,-71.101,-177.075,8.143,148.734
C03452=1155.159,287.139,-71.131,-177.072,8.146,148.734
C03453=1155.155,287.415,-71.164,-177.068,8.149,148.734
C03454=1155.150,287.689,-71.197,-177.066,8.153,148.734
C03455=1155.145,287.965,-71.230,-177.063,8.156,148.734
C03456=1155.141,288.240,-71.263,-177.060,8.159,148.734
C03457=1155.136,288.488,-71.293,-177.058,8.163,148.734
C03458=1155.132,288.736,-71.323,-177.055,8.166,148.734
C03459=1155.128,288.984,-71.353,-177.053,8.169,148.734
C03460=1155.123,289.232,-71.382,-177.049,8.173,148.734
C03461=1155.120,289.480,-71.412,-177.047,8.176,148.734
C03462=1155.115,289.729,-71.443,-177.044,8.179,148.734
C03463=1155.111,289.977,-71.473,-177.041,8.182,148.734
C03464=1155.107,290.225,-71.502,-177.039,8.185,148.734
C03465=1155.103,290.473,-71.533,-177.036,8.188,148.734
C03466=1155.098,290.721,-71.563,-177.034,8.191,148.734
C03467=1155.094,290.969,-71.593,-177.031,8.194,148.735
C03468=1155.090,291.218,-71.623,-177.029,8.197,148.735
C03469=1155.086,291.465,-71.653,-177.026,8.201,148.735
C03470=1155.081,291.714,-71.683,-177.023,8.204,148.735
C03471=1155.077,291.961,-71.713,-177.020,8.207,148.735
C03472=1155.073,292.210,-71.743,-177.018,8.211,148.735
C03473=1155.069,292.458,-71.774,-177.015,8.213,148.735
C03474=1155.064,292.707,-71.803,-177.013,8.217,148.735
C03475=1155.060,292.955,-71.834,-177.010,8.220,148.735
C03476=1155.056,293.202,-71.864,-177.008,8.223,148.735
C03477=1155.051,293.451,-71.894,-177.005,8.226,148.735
C03478=1155.048,293.699,-71.925,-177.002,8.230,148.735
C03479=1155.043,293.948,-71.955,-176.999,8.233,148.735
C03480=1155.039,294.195,-71.985,-176.996,8.236,148.735
C03481=1155.035,294.443,-72.015,-176.994,8.239,148.735
C03482=1155.031,294.691,-72.046,-176.991,8.242,148.735
C03483=1155.026,294.939,-72.075,-176.989,8.245,148.736
C03484=1155.022,295.188,-72.107,-176.986,8.248,148.735
C03485=1155.018,295.436,-72.137,-176.984,8.252,148.736
C03486=1155.014,295.684,-72.167,-176.981,8.255,148.736
C03487=1155.009,295.932,-72.198,-176.978,8.259,148.736
C03488=1155.006,296.180,-72.228,-176.976,8.262,148.736
C03489=1155.001,296.428,-72.259,-176.973,8.265,148.736
C03490=1154.997,296.676,-72.289,-176.971,8.268,148.736
C03491=1154.992,296.925,-72.319,-176.968,8.271,148.736
C03492=1154.988,297.172,-72.349,-176.965,8.274,148.736
C03493=1154.984,297.421,-72.380,-176.963,8.278,148.736
C03494=1154.980,297.669,-72.411,-176.960,8.281,148.736
C03495=1154.976,297.917,-72.441,-176.957,8.284,148.736
C03496=1154.971,298.165,-72.472,-176.955,8.287,148.736
C03497=1154.968,298.413,-72.503,-176.952,8.291,148.737
C03498=1154.963,298.661,-72.533,-176.950,8.294,148.737
C03499=1154.958,298.909,-72.563,-176.947,8.297,148.737
C03500=1154.955,299.158,-72.594,-176.944,8.301,148.737
C03501=1154.951,299.406,-72.625,-176.942,8.304,148.737
C03502=1154.946,299.654,-72.655,-176.939,8.307,148.737
C03503=1154.942,299.901,-72.686,-176.937,8.310,148.737
C03504=1154.938,300.150,-72.717,-176.934,8.313,148.737
C03505=1154.933,300.398,-72.747,-176.932,8.316,148.737
C03506=1154.929,300.646,-72.778,-176.928,8.320,148.737
C03507=1154.926,300.894,-72.809,-176.926,8.323,148.737
C03508=1154.921,301.142,-72.840,-176.923,8.326,148.737
C03509=1154.916,301.390,-72.870,-176.921,8.330,148.738
C03510=1154.913,301.638,-72.902,-176.918,8.333,148.738
C03511=1154.909,301.886,-72.932,-176.916,8.336,148.738
C03512=1154.904,302.134,-72.963,-176.913,8.340,148.738
C03513=1154.900,302.382,-72.994,-176.910,8.343,148.738
C03514=1154.896,302.630,-73.025,-176.908,8.346,148.738
C03515=1154.892,302.878,-73.055,-176.905,8.349,148.738
C03516=1154.888,303.127,-73.086,-176.903,8.353,148.738
C03517=1154.883,303.375,-73.117,-176.899,8.356,148.738
C03518=1154.879,303.622,-73.149,-176.897,8.360,148.738
C03519=1154.875,303.871,-73.180,-176.895,8.363,148.739
C03520=1154.870,304.119,-73.210,-176.892,8.366,148.739
C03521=1154.867,304.367,-73.241,-176.890,8.369,148.739
C03522=1154.862,304.614,-73.272,-176.887,8.372,148.739
C03523=1154.858,304.862,-73.303,-176.884,8.376,148.739
C03524=1154.854,305.111,-73.334,-176.882,8.379,148.739
C03525=1154.849,305.359,-73.365,-176.879,8.382,148.739
C03526=1154.846,305.607,-73.397,-176.877,8.386,148.739
C03527=1154.841,305.855,-73.428,-176.874,8.389,148.739
C03528=1154.836,306.103,-73.458,-176.871,8.393,148.740
C03529=1154.833,306.351,-73.490,-176.869,8.396,148.740
C03530=1154.828,306.599,-73.521,-176.866,8.399,148.740
C03531=1154.825,306.847,-73.552,-176.864,8.402,148.740
C03532=1154.820,307.095,-73.583,-176.861,8.405,148.740
C03533=1154.816,307.343,-73.614,-176.858,8.409,148.740
C03534=1154.812,307.591,-73.646,-176.856,8.413,148.740
C03535=1154.808,307.839,-73.677,-176.853,8.415,148.740
C03536=1154.803,308.087,-73.708,-176.851,8.419,148.740
C03537=1154.799,308.334,-73.739,-176.848,8.422,148.741
C03538=1154.795,308.583,-73.770,-176.845,8.426,148.741
C03539=1154.791,308.830,-73.802,-176.843,8.429,148.741
C03540=1154.787,309.079,-73.833,-176.840,8.432,148.741
C03541=1154.783,309.326,-73.864,-176.838,8.435,148.741
C03542=1154.779,309.575,-73.895,-176.835,8.439,148.741
C03543=1154.774,309.822,-73.927,-176.832,8.443,148.741
C03544=1154.770,310.071,-73.959,-176.830,8.446,148.741
C03545=1154.765,310.319,-73.990,-176.827,8.449,148.741
C03546=1154.761,310.567,-74.022,-176.825,8.452,148.742
C03547=1154.757,310.815,-74.053,-176.822,8.456,148.742
C03548=1154.753,311.063,-74.085,-176.819,8.459,148.742
C03549=1154.749,311.311,-74.116,-176.817,8.463,148.742
C03550=1154.745,311.559,-74.147,-176.814,8.465,148.742
C03551=1154.741,311.807,-74.179,-176.811,8.470,148.742
C03552=1154.736,312.055,-74.210,-176.809,8.473,148.742
C03553=1154.733,312.303,-74.242,-176.806,8.476,148.742
C03554=1154.728,312.550,-74.273,-176.804,8.479,148.743
C03555=1154.724,312.799,-74.306,-176.802,8.482,148.743
C03556=1154.720,313.047,-74.337,-176.798,8.486,148.743
C03557=1154.715,313.324,-74.372,-176.796,8.489,148.743
C03558=1154.711,313.602,-74.408,-176.793,8.494,148.743
C03559=1154.706,313.878,-74.443,-176.790,8.497,148.743
C03560=1154.702,314.156,-74.478,-176.787,8.501,148.744
C03561=1154.698,314.405,-74.510,-176.785,8.505,148.744
C03562=1154.693,314.652,-74.541,-176.782,8.508,148.744
C03563=1154.689,314.900,-74.573,-176.779,8.511,148.744
C03564=1154.685,315.148,-74.605,-176.777,8.515,148.744
C03565=1154.681,315.396,-74.637,-176.774,8.518,148.744
C03566=1154.677,315.644,-74.669,-176.771,8.521,148.744
C03567=1154.672,315.892,-74.700,-176.769,8.525,148.744
C03568=1154.668,316.140,-74.732,-176.766,8.529,148.745
C03569=1154.664,316.388,-74.764,-176.764,8.532,148.745
C03570=1154.660,316.635,-74.795,-176.761,8.535,148.745
C03571=1154.656,316.884,-74.828,-176.758,8.539,148.745
C03572=1154.652,317.132,-74.859,-176.756,8.542,148.745
C03573=1154.648,317.379,-74.891,-176.754,8.546,148.745
C03574=1154.643,317.627,-74.923,-176.751,8.549,148.746
C03575=1154.639,317.875,-74.955,-176.748,8.553,148.746
C03576=1154.636,318.124,-74.987,-176.746,8.556,148.746
C03577=1154.631,318.371,-75.019,-176.743,8.559,148.746
C03578=1154.627,318.619,-75.051,-176.741,8.562,148.746
C03579=1154.623,318.867,-75.083,-176.738,8.566,148.746
C03580=1154.618,319.115,-75.115,-176.735,8.569,148.746
C03581=1154.614,319.363,-75.147,-176.733,8.573,148.747
C03582=1154.611,319.611,-75.179,-176.730,8.577,148.747
C03583=1154.606,319.859,-75.211,-176.728,8.580,148.747
C03584=1154.602,320.106,-75.243,-176.725,8.583,148.747
C03585=1154.598,320.354,-75.276,-176.723,8.586,148.747
C03586=1154.594,320.602,-75.307,-176.720,8.590,148.747
C03587=1154.590,320.850,-75.339,-176.718,8.594,148.748
C03588=1154.585,321.098,-75.371,-176.715,8.597,148.748
C03589=1154.582,321.346,-75.403,-176.712,8.601,148.748
C03590=1154.578,321.594,-75.436,-176.710,8.604,148.748
C03591=1154.574,321.842,-75.468,-176.707,8.607,148.748
C03592=1154.569,322.090,-75.500,-176.705,8.611,148.748
C03593=1154.565,322.338,-75.532,-176.702,8.615,148.749
C03594=1154.561,322.585,-75.565,-176.700,8.618,148.749
C03595=1154.557,322.833,-75.597,-176.697,8.621,148.749
C03596=1154.553,323.082,-75.630,-176.694,8.625,148.749
C03597=1154.549,323.328,-75.662,-176.692,8.628,148.749
C03598=1154.544,323.577,-75.694,-176.690,8.632,148.750
C03599=1154.541,323.825,-75.726,-176.687,8.636,148.750
C03600=1154.537,324.073,-75.759,-176.684,8.639,148.750
C03601=1154.533,324.321,-75.791,-176.682,8.642,148.750
C03602=1154.528,324.569,-75.824,-176.679,8.645,148.750
C03603=1154.524,324.816,-75.856,-176.676,8.649,148.750
C03604=1154.520,325.064,-75.888,-176.674,8.653,148.751
C03605=1154.517,325.311,-75.921,-176.672,8.656,148.751
C03606=1154.512,325.560,-75.953,-176.669,8.660,148.751
C03607=1154.508,325.808,-75.986,-176.667,8.663,148.751
C03608=1154.504,326.056,-76.018,-176.664,8.666,148.751
C03609=1154.500,326.304,-76.051,-176.661,8.670,148.751
C03610=1154.496,326.551,-76.083,-176.659,8.674,148.752
C03611=1154.491,326.799,-76.115,-176.656,8.677,148.752
C03612=1154.487,327.047,-76.148,-176.653,8.681,148.752
C03613=1154.484,327.295,-76.180,-176.651,8.684,148.752
C03614=1154.479,327.542,-76.213,-176.649,8.687,148.752
C03615=1154.475,327.791,-76.246,-176.646,8.692,148.753
C03616=1154.472,328.038,-76.278,-176.644,8.695,148.753
C03617=1154.467,328.286,-76.312,-176.641,8.698,148.753
C03618=1154.463,328.534,-76.344,-176.638,8.702,148.753
C03619=1154.459,328.782,-76.377,-176.636,8.706,148.754
C03620=1154.455,329.029,-76.409,-176.633,8.708,148.753
C03621=1154.450,329.277,-76.442,-176.630,8.713,148.754
C03622=1154.446,329.525,-76.475,-176.628,8.716,148.754
C03623=1154.442,329.773,-76.507,-176.626,8.719,148.754
C03624=1154.438,330.021,-76.540,-176.623,8.723,148.754
C03625=1154.434,330.268,-76.573,-176.621,8.726,148.755
C03626=1154.430,330.516,-76.606,-176.618,8.730,148.755
C03627=1154.426,330.764,-76.639,-176.615,8.734,148.755
C03628=1154.422,331.012,-76.671,-176.613,8.737,148.755
C03629=1154.418,331.260,-76.704,-176.611,8.740,148.755
C03630=1154.414,331.507,-76.738,-176.608,8.745,148.756
C03631=1154.410,331.756,-76.770,-176.606,8.748,148.756
C03632=1154.405,332.003,-76.803,-176.603,8.752,148.756
C03633=1154.401,332.251,-76.836,-176.600,8.755,148.756
C03634=1154.398,332.499,-76.869,-176.598,8.758,148.756
C03635=1154.394,332.746,-76.902,-176.595,8.763,148.757
C03636=1154.390,332.994,-76.935,-176.593,8.766,148.757
C03637=1154.385,333.242,-76.968,-176.590,8.769,148.757
C03638=1154.381,333.490,-77.001,-176.588,8.773,148.757
C03639=1154.377,333.738,-77.034,-176.585,8.776,148.758
C03640=1154.373,333.986,-77.067,-176.582,8.781,148.758
C03641=1154.369,334.233,-77.100,-176.580,8.784,148.758
C03642=1154.365,334.481,-77.133,-176.578,8.787,148.758
C03643=1154.361,334.728,-77.166,-176.575,8.791,148.758
C03644=1154.357,334.976,-77.199,-176.573,8.794,148.759
C03645=1154.353,335.224,-77.232,-176.570,8.798,148.759
C03646=1154.349,335.472,-77.265,-176.567,8.802,148.759
C03647=1154.345,335.720,-77.299,-176.565,8.805,148.759
C03648=1154.341,335.968,-77.332,-176.562,8.809,148.760
C03649=1154.337,336.215,-77.365,-176.560,8.813,148.760
C03650=1154.333,336.463,-77.398,-176.557,8.816,148.760
C03651=1154.329,336.711,-77.432,-176.555,8.820,148.760
C03652=1154.324,336.959,-77.465,-176.552,8.823,148.760
C03653=1154.320,337.206,-77.498,-176.549,8.827,148.761
C03654=1154.316,337.454,-77.531,-176.547,8.831,148.761
C03655=1154.312,337.701,-77.565,-176.545,8.834,148.761
C03656=1154.308,337.949,-77.598,-176.542,8.838,148.761
C03657=1154.305,338.197,-77.632,-176.540,8.841,148.762
C03658=1154.300,338.445,-77.665,-176.537,8.845,148.762
C03659=1154.296,338.693,-77.698,-176.534,8.849,148.762
C03660=1154.292,338.941,-77.731,-176.532,8.852,148.762
C03661=1154.287,339.220,-77.769,-176.530,8.856,148.763
